LIN {X 0,Y 446.461,Z 349.006,A -85,B 0,C 180,E1 -8845.153,E2 -8845.153} C_VEL
LIN {X 0,Y 446.623,Z 343.213,A -85,B 0,C 180,E1 -8848.209,E2 -8848.209} C_VEL
LIN {X 0,Y 446.792,Z 337.441,A -85,B 0,C 180,E1 -8851.271,E2 -8851.271} C_VEL
LIN {X 0,Y 446.944,Z 331.506,A -85,B 0,C 180,E1 -8854.478,E2 -8854.478} C_VEL
LIN {X 0,Y 446.761,Z 327.48,A -85,B 0,C 180,E1 -8856.711,E2 -8856.711} C_VEL
LIN {X 0,Y 446.448,Z 325.193,A -85,B 0,C 180,E1 -8858.083,E2 -8858.083} C_VEL
LIN {X 0,Y 446.427,Z 325.192,A -85,B 0,C 180,E1 -8861.392,E2 -8861.392} C_VEL
LIN {X 0,Y 446.459,Z 325.185,A -85,B 0,C 180,E1 -8865.103,E2 -8865.103} C_VEL
LIN {X 0,Y 446.427,Z 325.19,A -85,B 0,C 180,E1 -8868.607,E2 -8868.607} C_VEL
LIN {X 0,Y 446.446,Z 325.238,A -85,B 0,C 180,E1 -8872.195,E2 -8872.195} C_VEL
LIN {X 0,Y 447.33,Z 330.595,A -85,B 0,C 180,E1 -8874.456,E2 -8874.456} C_VEL
LIN {X 0,Y 447.36,Z 335.572,A -85,B 0,C 180,E1 -8876.642,E2 -8876.642} C_VEL
LIN {X 0,Y 447.289,Z 341.416,A -85,B 0,C 180,E1 -8879.291,E2 -8879.291} C_VEL
LIN {X 0,Y 447.134,Z 348.904,A -85,B 0,C 180,E1 -8882.881,E2 -8882.881} C_VEL
LIN {X 0,Y 447.053,Z 356.132,A -85,B 0,C 180,E1 -8886.365,E2 -8886.365} C_VEL
LIN {X 0,Y 447.035,Z 362.429,A -85,B 0,C 180,E1 -8889.282,E2 -8889.282} C_VEL
LIN {X 0,Y 447.062,Z 369.132,A -85,B 0,C 180,E1 -8892.147,E2 -8892.147} C_VEL
LIN {X 0,Y 447.15,Z 373.659,A -85,B 0,C 180,E1 -8893.935,E2 -8893.935} C_VEL
LIN {X 0,Y 450.462,Z 384.816,A -85,B 0,C 180,E1 -8894.365,E2 -8894.365} C_VEL
LIN {X 0,Y 450.278,Z 397.037,A -85,B 0,C 180,E1 -8894.843,E2 -8894.843} C_VEL
LIN {X 0,Y 450.162,Z 402.389,A -85,B 0,C 180,E1 -8895.109,E2 -8895.109} C_VEL
LIN {X 0,Y 449.369,Z 407.874,A -85,B 0,C 180,E1 -8895.39,E2 -8895.39} C_VEL
LIN {X 0,Y 446.264,Z 416.577,A -85,B 0,C 180,E1 -8895.849,E2 -8895.849} C_VEL
LIN {X 0,Y 443.161,Z 424.955,A -85,B 0,C 180,E1 -8896.399,E2 -8896.399} C_VEL
LIN {X 0,Y 442.371,Z 429.793,A -85,B 0,C 180,E1 -8896.82,E2 -8896.82} C_VEL
LIN {X 0,Y 441.837,Z 439.223,A -85,B 0,C 180,E1 -8897.831,E2 -8897.831} C_VEL
LIN {X 0,Y 441.38,Z 447.936,A -85,B 0,C 180,E1 -8898.983,E2 -8898.983} C_VEL
LIN {X 0,Y 440.744,Z 456.447,A -85,B 0,C 180,E1 -8900.36,E2 -8900.36} C_VEL
LIN {X 0,Y 440.416,Z 463.236,A -85,B 0,C 180,E1 -8901.741,E2 -8901.741} C_VEL
LIN {X 0,Y 440.057,Z 468.639,A -85,B 0,C 180,E1 -8903.119,E2 -8903.119} C_VEL
LIN {X 0,Y 439.605,Z 472.902,A -85,B 0,C 180,E1 -8904.493,E2 -8904.493} C_VEL
LIN {X 0,Y 439.523,Z 475.12,A -85,B 0,C 180,E1 -8905.412,E2 -8905.412} C_VEL
LIN {X 0,Y 439.525,Z 476.919,A -85,B 0,C 180,E1 -8906.331,E2 -8906.331} C_VEL
LIN {X 0,Y 439.382,Z 478.317,A -85,B 0,C 180,E1 -8907.247,E2 -8907.247} C_VEL
LIN {X 0,Y 439.289,Z 479.89,A -85,B 0,C 180,E1 -8909.081,E2 -8909.081} C_VEL
LIN {X 0,Y 439.262,Z 480.124,A -85,B 0,C 180,E1 -8909.998,E2 -8909.998} C_VEL
LIN {X 0,Y 439.328,Z 479.368,A -85,B 0,C 180,E1 -8911.831,E2 -8911.831} C_VEL
LIN {X 0,Y 439.568,Z 477.087,A -85,B 0,C 180,E1 -8913.664,E2 -8913.664} C_VEL
LIN {X 0,Y 439.664,Z 474.304,A -85,B 0,C 180,E1 -8915.041,E2 -8915.041} C_VEL
LIN {X 0,Y 439.899,Z 470.504,A -85,B 0,C 180,E1 -8916.419,E2 -8916.419} C_VEL
LIN {X 0,Y 440.256,Z 465.229,A -85,B 0,C 180,E1 -8917.878,E2 -8917.878} C_VEL
LIN {X 0,Y 440.681,Z 458.173,A -85,B 0,C 180,E1 -8919.406,E2 -8919.406} C_VEL
LIN {X 0,Y 441.253,Z 450.147,A -85,B 0,C 180,E1 -8920.784,E2 -8920.784} C_VEL
LIN {X 0,Y 441.749,Z 441.869,A -85,B 0,C 180,E1 -8921.934,E2 -8921.934} C_VEL
LIN {X 0,Y 442.246,Z 431.688,A -85,B 0,C 180,E1 -8923.086,E2 -8923.086} C_VEL
LIN {X 0,Y 442.817,Z 421.179,A -85,B 0,C 180,E1 -8924.037,E2 -8924.037} C_VEL
LIN {X 0,Y 443.136,Z 410.38,A -85,B 0,C 180,E1 -8924.815,E2 -8924.815} C_VEL
LIN {X 0,Y 443.557,Z 397.678,A -85,B 0,C 180,E1 -8925.506,E2 -8925.506} C_VEL
LIN {X 0,Y 443.583,Z 385.861,A -85,B 0,C 180,E1 -8925.977,E2 -8925.977} C_VEL
LIN {X 0,Y 440.246,Z 374.666,A -85,B 0,C 180,E1 -8926.418,E2 -8926.418} C_VEL
LIN {X 0,Y 440.106,Z 366.794,A -85,B 0,C 180,E1 -8929.591,E2 -8929.591} C_VEL
LIN {X 0,Y 440.115,Z 359.098,A -85,B 0,C 180,E1 -8933.028,E2 -8933.028} C_VEL
LIN {X 0,Y 440.174,Z 351.628,A -85,B 0,C 180,E1 -8936.604,E2 -8936.604} C_VEL
LIN {X 0,Y 440.283,Z 345.234,A -85,B 0,C 180,E1 -8939.656,E2 -8939.656} C_VEL
LIN {X 0,Y 440.425,Z 338.39,A -85,B 0,C 180,E1 -8942.854,E2 -8942.854} C_VEL
LIN {X 0,Y 440.417,Z 332.314,A -85,B 0,C 180,E1 -8945.527,E2 -8945.527} C_VEL
LIN {X 0,Y 439.411,Z 326.272,A -85,B 0,C 180,E1 -8948.099,E2 -8948.099} C_VEL
LIN {X 0,Y 439.368,Z 326.07,A -85,B 0,C 180,E1 -8951.253,E2 -8951.253} C_VEL
LIN {X 0,Y 439.387,Z 326.066,A -85,B 0,C 180,E1 -8954.727,E2 -8954.727} C_VEL
LIN {X 0,Y 439.397,Z 326.062,A -85,B 0,C 180,E1 -8957.795,E2 -8957.795} C_VEL
LIN {X 0,Y 439.438,Z 326.06,A -85,B 0,C 180,E1 -8960.228,E2 -8960.228} C_VEL
LIN {X 0,Y 439.359,Z 326.071,A -85,B 0,C 180,E1 -8963.711,E2 -8963.711} C_VEL
LIN {X 0,Y 439.353,Z 326.069,A -85,B 0,C 180,E1 -8967.052,E2 -8967.052} C_VEL
LIN {X 0,Y 439.362,Z 326.064,A -85,B 0,C 180,E1 -8970.272,E2 -8970.272} C_VEL
LIN {X 0,Y 439.409,Z 326.056,A -85,B 0,C 180,E1 -8973.395,E2 -8973.395} C_VEL
LIN {X 0,Y 439.378,Z 326.063,A -85,B 0,C 180,E1 -8976.429,E2 -8976.429} C_VEL
LIN {X 0,Y 439.392,Z 326.067,A -85,B 0,C 180,E1 -8979.397,E2 -8979.397} C_VEL
LIN {X 0,Y 439.407,Z 326.059,A -85,B 0,C 180,E1 -8982.308,E2 -8982.308} C_VEL
LIN {X 0,Y 439.425,Z 326.054,A -85,B 0,C 180,E1 -8985.173,E2 -8985.173} C_VEL
LIN {X 0,Y 439.493,Z 326.052,A -85,B 0,C 180,E1 -8988.001,E2 -8988.001} C_VEL
LIN {X 0,Y 439.525,Z 326.045,A -85,B 0,C 180,E1 -8991.725,E2 -8991.725} C_VEL
LIN {X 0,Y 439.599,Z 326.034,A -85,B 0,C 180,E1 -8994.495,E2 -8994.495} C_VEL
LIN {X 0,Y 439.608,Z 326.037,A -85,B 0,C 180,E1 -8998.167,E2 -8998.167} C_VEL
LIN {X 0,Y 439.736,Z 326.017,A -85,B 0,C 180,E1 -9000,E2 -9000} C_VEL
LIN {X 0,Y 439.642,Z 326.034,A -85,B 0,C 180,E1 -9002.748,E2 -9002.748} C_VEL
LIN {X 0,Y 439.599,Z 326.037,A -85,B 0,C 180,E1 -9006.425,E2 -9006.425} C_VEL
LIN {X 0,Y 439.478,Z 326.056,A -85,B 0,C 180,E1 -9009.202,E2 -9009.202} C_VEL
LIN {X 0,Y 439.479,Z 326.057,A -85,B 0,C 180,E1 -9012.727,E2 -9012.727} C_VEL
LIN {X 0,Y 439.437,Z 326.062,A -85,B 0,C 180,E1 -9016.356,E2 -9016.356} C_VEL
LIN {X 0,Y 439.412,Z 326.065,A -85,B 0,C 180,E1 -9019.625,E2 -9019.625} C_VEL
LIN {X 0,Y 439.361,Z 326.068,A -85,B 0,C 180,E1 -9022.575,E2 -9022.575} C_VEL
LIN {X 0,Y 439.383,Z 326.065,A -85,B 0,C 180,E1 -9025.586,E2 -9025.586} C_VEL
LIN {X 0,Y 439.394,Z 326.066,A -85,B 0,C 180,E1 -9028.675,E2 -9028.675} C_VEL
LIN {X 0,Y 439.348,Z 326.072,A -85,B 0,C 180,E1 -9032.032,E2 -9032.032} C_VEL
LIN {X 0,Y 439.375,Z 326.069,A -85,B 0,C 180,E1 -9035.342,E2 -9035.342} C_VEL
LIN {X 0,Y 439.368,Z 326.069,A -85,B 0,C 180,E1 -9038.596,E2 -9038.596} C_VEL
LIN {X 0,Y 439.368,Z 326.062,A -85,B 0,C 180,E1 -9041.259,E2 -9041.259} C_VEL
LIN {X 0,Y 439.371,Z 326.248,A -85,B 0,C 180,E1 -9042.947,E2 -9042.947} C_VEL
LIN {X 0,Y 442.981,Z 337.856,A -85,B 0,C 180,E1 -9046.208,E2 -9046.208} C_VEL
LIN {X 0,Y 446.307,Z 349.009,A -85,B 0,C 180,E1 -9049.1,E2 -9049.1} C_VEL
LIN {X 0,Y 449.627,Z 361.072,A -85,B 0,C 180,E1 -9051.982,E2 -9051.982} C_VEL
LIN {X 0,Y 450.25,Z 364.591,A -85,B 0,C 180,E1 -9052.755,E2 -9052.755} C_VEL
LIN {X 0,Y 448.272,Z 381.256,A -85,B 0,C 180,E1 -9055.841,E2 -9055.841} C_VEL
LIN {X 0,Y 446.343,Z 400.241,A -85,B 0,C 180,E1 -9059.224,E2 -9059.224} C_VEL
LIN {X 0,Y 444.714,Z 418.995,A -85,B 0,C 180,E1 -9062.434,E2 -9062.434} C_VEL
LIN {X 0,Y 448.564,Z 438.005,A -85,B 0,C 180,E1 -9063.026,E2 -9063.026} C_VEL
LIN {X 0,Y 450.842,Z 449.868,A -85,B 0,C 180,E1 -9063.456,E2 -9063.456} C_VEL
LIN {X 0,Y 450.018,Z 466.755,A -85,B 0,C 180,E1 -9064.027,E2 -9064.027} C_VEL
LIN {X 0,Y 448.92,Z 482.813,A -85,B 0,C 180,E1 -9064.751,E2 -9064.751} C_VEL
LIN {X 0,Y 447.777,Z 498.534,A -85,B 0,C 180,E1 -9065.655,E2 -9065.655} C_VEL
LIN {X 0,Y 446.46,Z 513.475,A -85,B 0,C 180,E1 -9066.705,E2 -9066.705} C_VEL
LIN {X 0,Y 445.229,Z 527.23,A -85,B 0,C 180,E1 -9067.863,E2 -9067.863} C_VEL
LIN {X 0,Y 443.946,Z 540.246,A -85,B 0,C 180,E1 -9069.164,E2 -9069.164} C_VEL
LIN {X 0,Y 442.819,Z 551.987,A -85,B 0,C 180,E1 -9070.534,E2 -9070.534} C_VEL
LIN {X 0,Y 441.677,Z 563.981,A -85,B 0,C 180,E1 -9072.166,E2 -9072.166} C_VEL
LIN {X 0,Y 440.861,Z 574.252,A -85,B 0,C 180,E1 -9073.804,E2 -9073.804} C_VEL
LIN {X 0,Y 439.913,Z 584.129,A -85,B 0,C 180,E1 -9075.666,E2 -9075.666} C_VEL
LIN {X 0,Y 439.314,Z 592.39,A -85,B 0,C 180,E1 -9077.521,E2 -9077.521} C_VEL
LIN {X 0,Y 438.849,Z 599.352,A -85,B 0,C 180,E1 -9079.39,E2 -9079.39} C_VEL
LIN {X 0,Y 438.557,Z 604.908,A -85,B 0,C 180,E1 -9081.246,E2 -9081.246} C_VEL
LIN {X 0,Y 438.487,Z 608.25,A -85,B 0,C 180,E1 -9082.636,E2 -9082.636} C_VEL
LIN {X 0,Y 438.325,Z 611.637,A -85,B 0,C 180,E1 -9084.482,E2 -9084.482} C_VEL
LIN {X 0,Y 438.232,Z 614.093,A -85,B 0,C 180,E1 -9086.324,E2 -9086.324} C_VEL
LIN {X 0,Y 438.267,Z 615.479,A -85,B 0,C 180,E1 -9088.164,E2 -9088.164} C_VEL
LIN {X 0,Y 438.201,Z 616,A -85,B 0,C 180,E1 -9090.002,E2 -9090.002} C_VEL
LIN {X 0,Y 438.268,Z 615.475,A -85,B 0,C 180,E1 -9091.84,E2 -9091.84} C_VEL
LIN {X 0,Y 438.233,Z 614.087,A -85,B 0,C 180,E1 -9093.68,E2 -9093.68} C_VEL
LIN {X 0,Y 438.328,Z 611.629,A -85,B 0,C 180,E1 -9095.523,E2 -9095.523} C_VEL
LIN {X 0,Y 438.491,Z 608.248,A -85,B 0,C 180,E1 -9097.369,E2 -9097.369} C_VEL
LIN {X 0,Y 438.61,Z 603.623,A -85,B 0,C 180,E1 -9099.222,E2 -9099.222} C_VEL
LIN {X 0,Y 438.95,Z 597.704,A -85,B 0,C 180,E1 -9101.079,E2 -9101.079} C_VEL
LIN {X 0,Y 439.462,Z 590.425,A -85,B 0,C 180,E1 -9102.94,E2 -9102.94} C_VEL
LIN {X 0,Y 440.115,Z 581.588,A -85,B 0,C 180,E1 -9104.805,E2 -9104.805} C_VEL
LIN {X 0,Y 440.914,Z 572.495,A -85,B 0,C 180,E1 -9106.437,E2 -9106.437} C_VEL
LIN {X 0,Y 441.815,Z 561.902,A -85,B 0,C 180,E1 -9108.072,E2 -9108.072} C_VEL
LIN {X 0,Y 442.998,Z 549.4,A -85,B 0,C 180,E1 -9109.704,E2 -9109.704} C_VEL
LIN {X 0,Y 444.234,Z 536.263,A -85,B 0,C 180,E1 -9111.155,E2 -9111.155} C_VEL
LIN {X 0,Y 445.561,Z 521.959,A -85,B 0,C 180,E1 -9112.491,E2 -9112.491} C_VEL
LIN {X 0,Y 446.849,Z 507.165,A -85,B 0,C 180,E1 -9113.646,E2 -9113.646} C_VEL
LIN {X 0,Y 448.088,Z 491.339,A -85,B 0,C 180,E1 -9114.666,E2 -9114.666} C_VEL
LIN {X 0,Y 449.103,Z 476.791,A -85,B 0,C 180,E1 -9115.429,E2 -9115.429} C_VEL
LIN {X 0,Y 449.967,Z 461.122,A -85,B 0,C 180,E1 -9116.073,E2 -9116.073} C_VEL
LIN {X 0,Y 450.451,Z 448.549,A -85,B 0,C 180,E1 -9116.483,E2 -9116.483} C_VEL
LIN {X 0,Y 446.474,Z 429.842,A -85,B 0,C 180,E1 -9117.127,E2 -9117.127} C_VEL
LIN {X 0,Y 444.442,Z 417.956,A -85,B 0,C 180,E1 -9117.482,E2 -9117.482} C_VEL
LIN {X 0,Y 445.968,Z 398.339,A -85,B 0,C 180,E1 -9120.81,E2 -9120.81} C_VEL
LIN {X 0,Y 447.911,Z 381.252,A -85,B 0,C 180,E1 -9123.963,E2 -9123.963} C_VEL
LIN {X 0,Y 449.866,Z 369.238,A -85,B 0,C 180,E1 -9126.418,E2 -9126.418} C_VEL
LIN {X 0,Y 450.593,Z 364.614,A -85,B 0,C 180,E1 -9127.468,E2 -9127.468} C_VEL
LIN {X 0,Y 449.805,Z 360.335,A -85,B 0,C 180,E1 -9128.683,E2 -9128.683} C_VEL
LIN {X 0,Y 448.275,Z 354.936,A -85,B 0,C 180,E1 -9130.543,E2 -9130.543} C_VEL
LIN {X 0,Y 446.832,Z 350.314,A -85,B 0,C 180,E1 -9132.559,E2 -9132.559} C_VEL
LIN {X 0,Y 445.545,Z 346.703,A -85,B 0,C 180,E1 -9134.78,E2 -9134.78} C_VEL
LIN {X 0,Y 444.874,Z 344.812,A -85,B 0,C 180,E1 -9136.612,E2 -9136.612} C_VEL
LIN {X 0,Y 444.45,Z 343.921,A -85,B 0,C 180,E1 -9138.384,E2 -9138.384} C_VEL
LIN {X 0,Y 444.133,Z 344.024,A -85,B 0,C 180,E1 -9140.731,E2 -9140.731} C_VEL
LIN {X 0,Y 444.01,Z 345.321,A -85,B 0,C 180,E1 -9143.024,E2 -9143.024} C_VEL
LIN {X 0,Y 443.891,Z 346.316,A -85,B 0,C 180,E1 -9144.14,E2 -9144.14} C_VEL
LIN {X 0,Y 443.269,Z 348.846,A -85,B 0,C 180,E1 -9146.295,E2 -9146.295} C_VEL
LIN {X 0,Y 442.41,Z 353.265,A -85,B 0,C 180,E1 -9149.447,E2 -9149.447} C_VEL
LIN {X 0,Y 441.782,Z 358.656,A -85,B 0,C 180,E1 -9152.984,E2 -9152.984} C_VEL
LIN {X 0,Y 441.41,Z 362.771,A -85,B 0,C 180,E1 -9155.546,E2 -9155.546} C_VEL
LIN {X 0,Y 441.086,Z 367.633,A -85,B 0,C 180,E1 -9158.502,E2 -9158.502} C_VEL
LIN {X 0,Y 440.69,Z 373.409,A -85,B 0,C 180,E1 -9161.882,E2 -9161.882} C_VEL
LIN {X 0,Y 440.661,Z 374.052,A -85,B 0,C 180,E1 -9162.26,E2 -9162.26} C_VEL
LIN {X 0,Y 445.876,Z 388.81,A -85,B 0,C 180,E1 -9163.25,E2 -9163.25} C_VEL
LIN {X 0,Y 446.258,Z 389.984,A -85,B 0,C 180,E1 -9163.332,E2 -9163.332} C_VEL
LIN {X 0,Y 445.506,Z 404.424,A -85,B 0,C 180,E1 -9164.133,E2 -9164.133} C_VEL
LIN {X 0,Y 444.724,Z 416.942,A -85,B 0,C 180,E1 -9165.017,E2 -9165.017} C_VEL
LIN {X 0,Y 443.894,Z 428.51,A -85,B 0,C 180,E1 -9166.028,E2 -9166.028} C_VEL
LIN {X 0,Y 443.133,Z 439.164,A -85,B 0,C 180,E1 -9167.172,E2 -9167.172} C_VEL
LIN {X 0,Y 442.528,Z 447.959,A -85,B 0,C 180,E1 -9168.318,E2 -9168.318} C_VEL
LIN {X 0,Y 441.789,Z 456.684,A -85,B 0,C 180,E1 -9169.691,E2 -9169.691} C_VEL
LIN {X 0,Y 441.224,Z 464.001,A -85,B 0,C 180,E1 -9171.124,E2 -9171.124} C_VEL
LIN {X 0,Y 440.591,Z 470.283,A -85,B 0,C 180,E1 -9172.669,E2 -9172.669} C_VEL
LIN {X 0,Y 440.281,Z 474.558,A -85,B 0,C 180,E1 -9174.045,E2 -9174.045} C_VEL
LIN {X 0,Y 440.078,Z 477.764,A -85,B 0,C 180,E1 -9175.42,E2 -9175.42} C_VEL
LIN {X 0,Y 439.939,Z 479.386,A -85,B 0,C 180,E1 -9176.337,E2 -9176.337} C_VEL
LIN {X 0,Y 439.781,Z 480.56,A -85,B 0,C 180,E1 -9177.252,E2 -9177.252} C_VEL
LIN {X 0,Y 439.59,Z 481.33,A -85,B 0,C 180,E1 -9178.168,E2 -9178.168} C_VEL
LIN {X 0,Y 439.525,Z 481.683,A -85,B 0,C 180,E1 -9179.084,E2 -9179.084} C_VEL
LIN {X 0,Y 439.45,Z 481.649,A -85,B 0,C 180,E1 -9180,E2 -9180} C_VEL
LIN {X 0,Y 439.413,Z 481.201,A -85,B 0,C 180,E1 -9180.917,E2 -9180.917} C_VEL
LIN {X 0,Y 439.416,Z 480.322,A -85,B 0,C 180,E1 -9181.833,E2 -9181.833} C_VEL
LIN {X 0,Y 439.518,Z 479.036,A -85,B 0,C 180,E1 -9182.75,E2 -9182.75} C_VEL
LIN {X 0,Y 439.509,Z 476.345,A -85,B 0,C 180,E1 -9184.127,E2 -9184.127} C_VEL
LIN {X 0,Y 439.516,Z 472.663,A -85,B 0,C 180,E1 -9185.506,E2 -9185.506} C_VEL
LIN {X 0,Y 439.883,Z 467.862,A -85,B 0,C 180,E1 -9186.883,E2 -9186.883} C_VEL
LIN {X 0,Y 440.15,Z 460.779,A -85,B 0,C 180,E1 -9188.494,E2 -9188.494} C_VEL
LIN {X 0,Y 440.59,Z 453.141,A -85,B 0,C 180,E1 -9189.874,E2 -9189.874} C_VEL
LIN {X 0,Y 440.995,Z 443.74,A -85,B 0,C 180,E1 -9191.258,E2 -9191.258} C_VEL
LIN {X 0,Y 441.643,Z 433.185,A -85,B 0,C 180,E1 -9192.523,E2 -9192.523} C_VEL
LIN {X 0,Y 442.18,Z 421.281,A -85,B 0,C 180,E1 -9193.676,E2 -9193.676} C_VEL
LIN {X 0,Y 442.714,Z 409.036,A -85,B 0,C 180,E1 -9194.632,E2 -9194.632} C_VEL
LIN {X 0,Y 443.317,Z 396.509,A -85,B 0,C 180,E1 -9195.399,E2 -9195.399} C_VEL
LIN {X 0,Y 443.526,Z 384.753,A -85,B 0,C 180,E1 -9195.969,E2 -9195.969} C_VEL
LIN {X 0,Y 440.231,Z 370.942,A -85,B 0,C 180,E1 -9196.607,E2 -9196.607} C_VEL
LIN {X 0,Y 439.07,Z 366.227,A -85,B 0,C 180,E1 -9196.806,E2 -9196.806} C_VEL
LIN {X 0,Y 439.16,Z 360.671,A -85,B 0,C 180,E1 -9199.638,E2 -9199.638} C_VEL
LIN {X 0,Y 439.289,Z 354.989,A -85,B 0,C 180,E1 -9202.58,E2 -9202.58} C_VEL
LIN {X 0,Y 439.444,Z 349.231,A -85,B 0,C 180,E1 -9205.583,E2 -9205.583} C_VEL
LIN {X 0,Y 439.617,Z 343.434,A -85,B 0,C 180,E1 -9208.66,E2 -9208.66} C_VEL
LIN {X 0,Y 439.838,Z 336.984,A -85,B 0,C 180,E1 -9212.125,E2 -9212.125} C_VEL
LIN {X 0,Y 439.939,Z 331.552,A -85,B 0,C 180,E1 -9215.107,E2 -9215.107} C_VEL
LIN {X 0,Y 439.605,Z 327.454,A -85,B 0,C 180,E1 -9217.41,E2 -9217.41} C_VEL
LIN {X 0,Y 439.403,Z 326.069,A -85,B 0,C 180,E1 -9218.314,E2 -9218.314} C_VEL
LIN {X 0,Y 439.39,Z 326.069,A -85,B 0,C 180,E1 -9221.255,E2 -9221.255} C_VEL
LIN {X 0,Y 439.407,Z 326.062,A -85,B 0,C 180,E1 -9224.729,E2 -9224.729} C_VEL
LIN {X 0,Y 439.393,Z 326.067,A -85,B 0,C 180,E1 -9227.793,E2 -9227.793} C_VEL
LIN {X 0,Y 439.367,Z 326.071,A -85,B 0,C 180,E1 -9230.219,E2 -9230.219} C_VEL
LIN {X 0,Y 439.424,Z 326.156,A -85,B 0,C 180,E1 -9231.944,E2 -9231.944} C_VEL
LIN {X 0,Y 440.38,Z 332.057,A -85,B 0,C 180,E1 -9234.48,E2 -9234.48} C_VEL
LIN {X 0,Y 440.377,Z 338.112,A -85,B 0,C 180,E1 -9237.137,E2 -9237.137} C_VEL
LIN {X 0,Y 440.289,Z 343.279,A -85,B 0,C 180,E1 -9239.538,E2 -9239.538} C_VEL
LIN {X 0,Y 440.169,Z 350.428,A -85,B 0,C 180,E1 -9242.931,E2 -9242.931} C_VEL
LIN {X 0,Y 440.101,Z 357.804,A -85,B 0,C 180,E1 -9246.468,E2 -9246.468} C_VEL
LIN {X 0,Y 440.095,Z 364.282,A -85,B 0,C 180,E1 -9249.43,E2 -9249.43} C_VEL
LIN {X 0,Y 440.132,Z 371.194,A -85,B 0,C 180,E1 -9252.337,E2 -9252.337} C_VEL
LIN {X 0,Y 440.23,Z 374.625,A -85,B 0,C 180,E1 -9253.67,E2 -9253.67} C_VEL
LIN {X 0,Y 443.722,Z 386.858,A -85,B 0,C 180,E1 -9254.157,E2 -9254.157} C_VEL
LIN {X 0,Y 443.505,Z 399.298,A -85,B 0,C 180,E1 -9254.664,E2 -9254.664} C_VEL
LIN {X 0,Y 443.097,Z 411.668,A -85,B 0,C 180,E1 -9255.36,E2 -9255.36} C_VEL
LIN {X 0,Y 442.665,Z 423.158,A -85,B 0,C 180,E1 -9256.221,E2 -9256.221} C_VEL
LIN {X 0,Y 442.371,Z 429.793,A -85,B 0,C 180,E1 -9256.82,E2 -9256.82} C_VEL
LIN {X 0,Y 441.605,Z 434.491,A -85,B 0,C 180,E1 -9257.273,E2 -9257.273} C_VEL
LIN {X 0,Y 438.52,Z 441.99,A -85,B 0,C 180,E1 -9258.014,E2 -9258.014} C_VEL
LIN {X 0,Y 435.241,Z 448.977,A -85,B 0,C 180,E1 -9258.832,E2 -9258.832} C_VEL
LIN {X 0,Y 434.191,Z 452.875,A -85,B 0,C 180,E1 -9259.403,E2 -9259.403} C_VEL
LIN {X 0,Y 433.717,Z 459.935,A -85,B 0,C 180,E1 -9260.673,E2 -9260.673} C_VEL
LIN {X 0,Y 433.282,Z 466.931,A -85,B 0,C 180,E1 -9262.244,E2 -9262.244} C_VEL
LIN {X 0,Y 432.947,Z 471.261,A -85,B 0,C 180,E1 -9263.473,E2 -9263.473} C_VEL
LIN {X 0,Y 432.663,Z 475.144,A -85,B 0,C 180,E1 -9264.872,E2 -9264.872} C_VEL
LIN {X 0,Y 432.529,Z 477.995,A -85,B 0,C 180,E1 -9266.271,E2 -9266.271} C_VEL
LIN {X 0,Y 432.401,Z 479.39,A -85,B 0,C 180,E1 -9267.203,E2 -9267.203} C_VEL
LIN {X 0,Y 432.275,Z 480.967,A -85,B 0,C 180,E1 -9269.066,E2 -9269.066} C_VEL
LIN {X 0,Y 432.245,Z 481.201,A -85,B 0,C 180,E1 -9269.998,E2 -9269.998} C_VEL
LIN {X 0,Y 432.325,Z 480.443,A -85,B 0,C 180,E1 -9271.861,E2 -9271.861} C_VEL
LIN {X 0,Y 432.566,Z 478.162,A -85,B 0,C 180,E1 -9273.724,E2 -9273.724} C_VEL
LIN {X 0,Y 432.671,Z 475.379,A -85,B 0,C 180,E1 -9275.123,E2 -9275.123} C_VEL
LIN {X 0,Y 432.929,Z 471.577,A -85,B 0,C 180,E1 -9276.522,E2 -9276.522} C_VEL
LIN {X 0,Y 433.322,Z 466.192,A -85,B 0,C 180,E1 -9278.031,E2 -9278.031} C_VEL
LIN {X 0,Y 433.755,Z 459.245,A -85,B 0,C 180,E1 -9279.557,E2 -9279.557} C_VEL
LIN {X 0,Y 434.369,Z 451.214,A -85,B 0,C 180,E1 -9280.957,E2 -9280.957} C_VEL
LIN {X 0,Y 434.889,Z 442.933,A -85,B 0,C 180,E1 -9282.125,E2 -9282.125} C_VEL
LIN {X 0,Y 435.427,Z 432.747,A -85,B 0,C 180,E1 -9283.295,E2 -9283.295} C_VEL
LIN {X 0,Y 436.018,Z 422.191,A -85,B 0,C 180,E1 -9284.264,E2 -9284.264} C_VEL
LIN {X 0,Y 436.347,Z 411.426,A -85,B 0,C 180,E1 -9285.051,E2 -9285.051} C_VEL
LIN {X 0,Y 436.782,Z 398.712,A -85,B 0,C 180,E1 -9285.752,E2 -9285.752} C_VEL
LIN {X 0,Y 436.914,Z 387.614,A -85,B 0,C 180,E1 -9286.201,E2 -9286.201} C_VEL
LIN {X 0,Y 433.337,Z 375.627,A -85,B 0,C 180,E1 -9286.696,E2 -9286.696} C_VEL
LIN {X 0,Y 433.186,Z 367.618,A -85,B 0,C 180,E1 -9289.917,E2 -9289.917} C_VEL
LIN {X 0,Y 433.167,Z 359.766,A -85,B 0,C 180,E1 -9293.419,E2 -9293.419} C_VEL
LIN {X 0,Y 433.21,Z 352.242,A -85,B 0,C 180,E1 -9297.013,E2 -9297.013} C_VEL
LIN {X 0,Y 433.346,Z 345.558,A -85,B 0,C 180,E1 -9300.179,E2 -9300.179} C_VEL
LIN {X 0,Y 433.488,Z 338.514,A -85,B 0,C 180,E1 -9303.448,E2 -9303.448} C_VEL
LIN {X 0,Y 433.386,Z 333.134,A -85,B 0,C 180,E1 -9305.823,E2 -9305.823} C_VEL
LIN {X 0,Y 432.456,Z 327.729,A -85,B 0,C 180,E1 -9308.134,E2 -9308.134} C_VEL
LIN {X 0,Y 432.321,Z 326.949,A -85,B 0,C 180,E1 -9308.514,E2 -9308.514} C_VEL
LIN {X 0,Y 432.31,Z 326.949,A -85,B 0,C 180,E1 -9311.796,E2 -9311.796} C_VEL
LIN {X 0,Y 432.364,Z 326.94,A -85,B 0,C 180,E1 -9315.656,E2 -9315.656} C_VEL
LIN {X 0,Y 432.358,Z 326.942,A -85,B 0,C 180,E1 -9318.389,E2 -9318.389} C_VEL
LIN {X 0,Y 432.338,Z 326.943,A -85,B 0,C 180,E1 -9321.85,E2 -9321.85} C_VEL
LIN {X 0,Y 432.322,Z 326.946,A -85,B 0,C 180,E1 -9325.321,E2 -9325.321} C_VEL
LIN {X 0,Y 432.301,Z 326.949,A -85,B 0,C 180,E1 -9328.652,E2 -9328.652} C_VEL
LIN {X 0,Y 432.362,Z 326.94,A -85,B 0,C 180,E1 -9331.875,E2 -9331.875} C_VEL
LIN {X 0,Y 432.338,Z 326.943,A -85,B 0,C 180,E1 -9334.998,E2 -9334.998} C_VEL
LIN {X 0,Y 432.389,Z 326.937,A -85,B 0,C 180,E1 -9338.047,E2 -9338.047} C_VEL
LIN {X 0,Y 432.363,Z 326.937,A -85,B 0,C 180,E1 -9341.028,E2 -9341.028} C_VEL
LIN {X 0,Y 432.407,Z 326.933,A -85,B 0,C 180,E1 -9343.96,E2 -9343.96} C_VEL
LIN {X 0,Y 432.464,Z 326.927,A -85,B 0,C 180,E1 -9347.803,E2 -9347.803} C_VEL
LIN {X 0,Y 432.469,Z 326.922,A -85,B 0,C 180,E1 -9351.59,E2 -9351.59} C_VEL
LIN {X 0,Y 432.575,Z 326.909,A -85,B 0,C 180,E1 -9354.405,E2 -9354.405} C_VEL
LIN {X 0,Y 432.577,Z 326.912,A -85,B 0,C 180,E1 -9358.138,E2 -9358.138} C_VEL
LIN {X 0,Y 432.706,Z 326.893,A -85,B 0,C 180,E1 -9360,E2 -9360} C_VEL
LIN {X 0,Y 432.592,Z 326.912,A -85,B 0,C 180,E1 -9362.793,E2 -9362.793} C_VEL
LIN {X 0,Y 432.552,Z 326.914,A -85,B 0,C 180,E1 -9366.53,E2 -9366.53} C_VEL
LIN {X 0,Y 432.422,Z 326.936,A -85,B 0,C 180,E1 -9369.353,E2 -9369.353} C_VEL
LIN {X 0,Y 432.419,Z 326.936,A -85,B 0,C 180,E1 -9372.812,E2 -9372.812} C_VEL
LIN {X 0,Y 432.399,Z 326.937,A -85,B 0,C 180,E1 -9376.485,E2 -9376.485} C_VEL
LIN {X 0,Y 432.359,Z 326.942,A -85,B 0,C 180,E1 -9379.959,E2 -9379.959} C_VEL
LIN {X 0,Y 432.31,Z 326.948,A -85,B 0,C 180,E1 -9382.964,E2 -9382.964} C_VEL
LIN {X 0,Y 432.341,Z 326.942,A -85,B 0,C 180,E1 -9386.034,E2 -9386.034} C_VEL
LIN {X 0,Y 432.319,Z 326.945,A -85,B 0,C 180,E1 -9389.189,E2 -9389.189} C_VEL
LIN {X 0,Y 432.301,Z 326.95,A -85,B 0,C 180,E1 -9392.444,E2 -9392.444} C_VEL
LIN {X 0,Y 432.325,Z 326.947,A -85,B 0,C 180,E1 -9395.634,E2 -9395.634} C_VEL
LIN {X 0,Y 432.331,Z 326.945,A -85,B 0,C 180,E1 -9398.718,E2 -9398.718} C_VEL
LIN {X 0,Y 432.356,Z 326.989,A -85,B 0,C 180,E1 -9402.186,E2 -9402.186} C_VEL
LIN {X 0,Y 436.303,Z 340.009,A -85,B 0,C 180,E1 -9405.924,E2 -9405.924} C_VEL
LIN {X 0,Y 439.476,Z 350.623,A -85,B 0,C 180,E1 -9408.73,E2 -9408.73} C_VEL
LIN {X 0,Y 442.95,Z 363.118,A -85,B 0,C 180,E1 -9411.776,E2 -9411.776} C_VEL
LIN {X 0,Y 443.582,Z 366.816,A -85,B 0,C 180,E1 -9412.606,E2 -9412.606} C_VEL
LIN {X 0,Y 441.61,Z 382.484,A -85,B 0,C 180,E1 -9415.565,E2 -9415.565} C_VEL
LIN {X 0,Y 439.679,Z 399.756,A -85,B 0,C 180,E1 -9418.705,E2 -9418.705} C_VEL
LIN {X 0,Y 437.968,Z 418.244,A -85,B 0,C 180,E1 -9421.954,E2 -9421.954} C_VEL
LIN {X 0,Y 437.938,Z 418.769,A -85,B 0,C 180,E1 -9422.039,E2 -9422.039} C_VEL
LIN {X 0,Y 442.163,Z 439.816,A -85,B 0,C 180,E1 -9422.713,E2 -9422.713} C_VEL
LIN {X 0,Y 444.247,Z 450.914,A -85,B 0,C 180,E1 -9423.142,E2 -9423.142} C_VEL
LIN {X 0,Y 443.356,Z 467.342,A -85,B 0,C 180,E1 -9423.717,E2 -9423.717} C_VEL
LIN {X 0,Y 442.213,Z 483.385,A -85,B 0,C 180,E1 -9424.466,E2 -9424.466} C_VEL
LIN {X 0,Y 441.037,Z 498.747,A -85,B 0,C 180,E1 -9425.377,E2 -9425.377} C_VEL
LIN {X 0,Y 439.66,Z 513.596,A -85,B 0,C 180,E1 -9426.448,E2 -9426.448} C_VEL
LIN {X 0,Y 438.249,Z 528.407,A -85,B 0,C 180,E1 -9427.74,E2 -9427.74} C_VEL
LIN {X 0,Y 436.881,Z 541.658,A -85,B 0,C 180,E1 -9429.11,E2 -9429.11} C_VEL
LIN {X 0,Y 435.605,Z 554.514,A -85,B 0,C 180,E1 -9430.689,E2 -9430.689} C_VEL
LIN {X 0,Y 434.504,Z 565.789,A -85,B 0,C 180,E1 -9432.319,E2 -9432.319} C_VEL
LIN {X 0,Y 433.649,Z 575.801,A -85,B 0,C 180,E1 -9434.01,E2 -9434.01} C_VEL
LIN {X 0,Y 432.73,Z 585.335,A -85,B 0,C 180,E1 -9435.903,E2 -9435.903} C_VEL
LIN {X 0,Y 432.151,Z 593.307,A -85,B 0,C 180,E1 -9437.797,E2 -9437.797} C_VEL
LIN {X 0,Y 431.672,Z 599.854,A -85,B 0,C 180,E1 -9439.686,E2 -9439.686} C_VEL
LIN {X 0,Y 431.478,Z 605.236,A -85,B 0,C 180,E1 -9441.573,E2 -9441.573} C_VEL
LIN {X 0,Y 431.321,Z 609.872,A -85,B 0,C 180,E1 -9443.687,E2 -9443.687} C_VEL
LIN {X 0,Y 431.211,Z 612.499,A -85,B 0,C 180,E1 -9445.328,E2 -9445.328} C_VEL
LIN {X 0,Y 431.196,Z 614.537,A -85,B 0,C 180,E1 -9447.2,E2 -9447.2} C_VEL
LIN {X 0,Y 431.144,Z 615.545,A -85,B 0,C 180,E1 -9449.068,E2 -9449.068} C_VEL
LIN {X 0,Y 431.144,Z 615.543,A -85,B 0,C 180,E1 -9450.936,E2 -9450.936} C_VEL
LIN {X 0,Y 431.197,Z 614.528,A -85,B 0,C 180,E1 -9452.805,E2 -9452.805} C_VEL
LIN {X 0,Y 431.213,Z 612.475,A -85,B 0,C 180,E1 -9454.676,E2 -9454.676} C_VEL
LIN {X 0,Y 431.362,Z 609.364,A -85,B 0,C 180,E1 -9456.551,E2 -9456.551} C_VEL
LIN {X 0,Y 431.48,Z 605.152,A -85,B 0,C 180,E1 -9458.432,E2 -9458.432} C_VEL
LIN {X 0,Y 431.681,Z 599.705,A -85,B 0,C 180,E1 -9460.319,E2 -9460.319} C_VEL
LIN {X 0,Y 432.186,Z 593.071,A -85,B 0,C 180,E1 -9462.206,E2 -9462.206} C_VEL
LIN {X 0,Y 432.755,Z 584.97,A -85,B 0,C 180,E1 -9464.101,E2 -9464.101} C_VEL
LIN {X 0,Y 433.645,Z 575.275,A -85,B 0,C 180,E1 -9465.995,E2 -9465.995} C_VEL
LIN {X 0,Y 434.466,Z 565.057,A -85,B 0,C 180,E1 -9467.686,E2 -9467.686} C_VEL
LIN {X 0,Y 435.58,Z 553.533,A -85,B 0,C 180,E1 -9469.317,E2 -9469.317} C_VEL
LIN {X 0,Y 436.873,Z 540.446,A -85,B 0,C 180,E1 -9470.889,E2 -9470.889} C_VEL
LIN {X 0,Y 438.186,Z 526.797,A -85,B 0,C 180,E1 -9472.269,E2 -9472.269} C_VEL
LIN {X 0,Y 439.407,Z 513.028,A -85,B 0,C 180,E1 -9473.446,E2 -9473.446} C_VEL
LIN {X 0,Y 440.797,Z 497.2,A -85,B 0,C 180,E1 -9474.572,E2 -9474.572} C_VEL
LIN {X 0,Y 442.003,Z 481.35,A -85,B 0,C 180,E1 -9475.489,E2 -9475.489} C_VEL
LIN {X 0,Y 443.027,Z 465.567,A -85,B 0,C 180,E1 -9476.214,E2 -9476.214} C_VEL
LIN {X 0,Y 443.827,Z 450.008,A -85,B 0,C 180,E1 -9476.755,E2 -9476.755} C_VEL
LIN {X 0,Y 440.208,Z 432.566,A -85,B 0,C 180,E1 -9477.401,E2 -9477.401} C_VEL
LIN {X 0,Y 437.6,Z 417.592,A -85,B 0,C 180,E1 -9477.858,E2 -9477.858} C_VEL
LIN {X 0,Y 439.182,Z 399.211,A -85,B 0,C 180,E1 -9481.071,E2 -9481.071} C_VEL
LIN {X 0,Y 441.14,Z 383.445,A -85,B 0,C 180,E1 -9484.062,E2 -9484.062} C_VEL
LIN {X 0,Y 443.635,Z 369.506,A -85,B 0,C 180,E1 -9487.014,E2 -9487.014} C_VEL
LIN {X 0,Y 443.966,Z 366.752,A -85,B 0,C 180,E1 -9487.674,E2 -9487.674} C_VEL
LIN {X 0,Y 443.088,Z 362.344,A -85,B 0,C 180,E1 -9488.995,E2 -9488.995} C_VEL
LIN {X 0,Y 441.74,Z 357.562,A -85,B 0,C 180,E1 -9490.717,E2 -9490.717} C_VEL
LIN {X 0,Y 440.327,Z 353.07,A -85,B 0,C 180,E1 -9492.761,E2 -9492.761} C_VEL
LIN {X 0,Y 439.195,Z 349.885,A -85,B 0,C 180,E1 -9494.758,E2 -9494.758} C_VEL
LIN {X 0,Y 438.542,Z 348.055,A -85,B 0,C 180,E1 -9496.441,E2 -9496.441} C_VEL
LIN {X 0,Y 438.2,Z 347.243,A -85,B 0,C 180,E1 -9497.654,E2 -9497.654} C_VEL
LIN {X 0,Y 437.717,Z 346.791,A -85,B 0,C 180,E1 -9500.041,E2 -9500.041} C_VEL
LIN {X 0,Y 437.507,Z 347.599,A -85,B 0,C 180,E1 -9502.38,E2 -9502.38} C_VEL
LIN {X 0,Y 437.106,Z 349.437,A -85,B 0,C 180,E1 -9504.632,E2 -9504.632} C_VEL
LIN {X 0,Y 436.382,Z 352.037,A -85,B 0,C 180,E1 -9506.876,E2 -9506.876} C_VEL
LIN {X 0,Y 435.378,Z 357.244,A -85,B 0,C 180,E1 -9510.657,E2 -9510.657} C_VEL
LIN {X 0,Y 434.941,Z 360.882,A -85,B 0,C 180,E1 -9513.1,E2 -9513.1} C_VEL
LIN {X 0,Y 434.458,Z 365.669,A -85,B 0,C 180,E1 -9516.146,E2 -9516.146} C_VEL
LIN {X 0,Y 434.143,Z 370.539,A -85,B 0,C 180,E1 -9519.137,E2 -9519.137} C_VEL
LIN {X 0,Y 433.83,Z 375.1,A -85,B 0,C 180,E1 -9521.813,E2 -9521.813} C_VEL
LIN {X 0,Y 438.73,Z 388.37,A -85,B 0,C 180,E1 -9522.751,E2 -9522.751} C_VEL
LIN {X 0,Y 439.801,Z 392.243,A -85,B 0,C 180,E1 -9523.027,E2 -9523.027} C_VEL
LIN {X 0,Y 438.926,Z 407.104,A -85,B 0,C 180,E1 -9523.889,E2 -9523.889} C_VEL
LIN {X 0,Y 438.183,Z 418.024,A -85,B 0,C 180,E1 -9524.687,E2 -9524.687} C_VEL
LIN {X 0,Y 437.241,Z 430.479,A -85,B 0,C 180,E1 -9525.811,E2 -9525.811} C_VEL
LIN {X 0,Y 436.434,Z 440.956,A -85,B 0,C 180,E1 -9526.971,E2 -9526.971} C_VEL
LIN {X 0,Y 435.789,Z 449.66,A -85,B 0,C 180,E1 -9528.135,E2 -9528.135} C_VEL
LIN {X 0,Y 434.993,Z 458.259,A -85,B 0,C 180,E1 -9529.528,E2 -9529.528} C_VEL
LIN {X 0,Y 434.315,Z 466.258,A -85,B 0,C 180,E1 -9531.157,E2 -9531.157} C_VEL
LIN {X 0,Y 433.697,Z 471.72,A -85,B 0,C 180,E1 -9532.552,E2 -9532.552} C_VEL
LIN {X 0,Y 433.383,Z 475.951,A -85,B 0,C 180,E1 -9533.95,E2 -9533.95} C_VEL
LIN {X 0,Y 433.156,Z 479.115,A -85,B 0,C 180,E1 -9535.347,E2 -9535.347} C_VEL
LIN {X 0,Y 432.983,Z 480.705,A -85,B 0,C 180,E1 -9536.278,E2 -9536.278} C_VEL
LIN {X 0,Y 432.827,Z 481.84,A -85,B 0,C 180,E1 -9537.208,E2 -9537.208} C_VEL
LIN {X 0,Y 432.626,Z 482.578,A -85,B 0,C 180,E1 -9538.138,E2 -9538.138} C_VEL
LIN {X 0,Y 432.548,Z 482.908,A -85,B 0,C 180,E1 -9539.069,E2 -9539.069} C_VEL
LIN {X 0,Y 432.474,Z 482.85,A -85,B 0,C 180,E1 -9540,E2 -9540} C_VEL
LIN {X 0,Y 432.421,Z 482.371,A -85,B 0,C 180,E1 -9540.932,E2 -9540.932} C_VEL
LIN {X 0,Y 432.413,Z 481.468,A -85,B 0,C 180,E1 -9541.863,E2 -9541.863} C_VEL
LIN {X 0,Y 432.522,Z 480.143,A -85,B 0,C 180,E1 -9542.794,E2 -9542.794} C_VEL
LIN {X 0,Y 432.505,Z 477.407,A -85,B 0,C 180,E1 -9544.194,E2 -9544.194} C_VEL
LIN {X 0,Y 432.522,Z 473.666,A -85,B 0,C 180,E1 -9545.595,E2 -9545.595} C_VEL
LIN {X 0,Y 432.909,Z 468.8,A -85,B 0,C 180,E1 -9546.994,E2 -9546.994} C_VEL
LIN {X 0,Y 433.2,Z 461.633,A -85,B 0,C 180,E1 -9548.631,E2 -9548.631} C_VEL
LIN {X 0,Y 433.664,Z 453.919,A -85,B 0,C 180,E1 -9550.033,E2 -9550.033} C_VEL
LIN {X 0,Y 434.08,Z 444.457,A -85,B 0,C 180,E1 -9551.44,E2 -9551.44} C_VEL
LIN {X 0,Y 434.753,Z 433.834,A -85,B 0,C 180,E1 -9552.724,E2 -9552.724} C_VEL
LIN {X 0,Y 435.321,Z 421.868,A -85,B 0,C 180,E1 -9553.896,E2 -9553.896} C_VEL
LIN {X 0,Y 435.87,Z 409.643,A -85,B 0,C 180,E1 -9554.863,E2 -9554.863} C_VEL
LIN {X 0,Y 436.517,Z 397.04,A -85,B 0,C 180,E1 -9555.645,E2 -9555.645} C_VEL
LIN {X 0,Y 436.699,Z 386.028,A -85,B 0,C 180,E1 -9556.195,E2 -9556.195} C_VEL
LIN {X 0,Y 433.44,Z 372.182,A -85,B 0,C 180,E1 -9556.85,E2 -9556.85} C_VEL
LIN {X 0,Y 432.041,Z 366.611,A -85,B 0,C 180,E1 -9557.087,E2 -9557.087} C_VEL
LIN {X 0,Y 432.137,Z 361.016,A -85,B 0,C 180,E1 -9559.971,E2 -9559.971} C_VEL
LIN {X 0,Y 432.26,Z 355.25,A -85,B 0,C 180,E1 -9562.968,E2 -9562.968} C_VEL
LIN {X 0,Y 432.427,Z 349.449,A -85,B 0,C 180,E1 -9566.029,E2 -9566.029} C_VEL
LIN {X 0,Y 432.618,Z 343.596,A -85,B 0,C 180,E1 -9569.168,E2 -9569.168} C_VEL
LIN {X 0,Y 432.845,Z 337.633,A -85,B 0,C 180,E1 -9572.4,E2 -9572.4} C_VEL
LIN {X 0,Y 432.931,Z 333.601,A -85,B 0,C 180,E1 -9574.623,E2 -9574.623} C_VEL
LIN {X 0,Y 432.73,Z 329.508,A -85,B 0,C 180,E1 -9576.936,E2 -9576.936} C_VEL
LIN {X 0,Y 432.356,Z 326.947,A -85,B 0,C 180,E1 -9578.429,E2 -9578.429} C_VEL
LIN {X 0,Y 432.333,Z 326.947,A -85,B 0,C 180,E1 -9581.798,E2 -9581.798} C_VEL
LIN {X 0,Y 432.343,Z 326.943,A -85,B 0,C 180,E1 -9584.347,E2 -9584.347} C_VEL
LIN {X 0,Y 432.325,Z 326.948,A -85,B 0,C 180,E1 -9587.016,E2 -9587.016} C_VEL
LIN {X 0,Y 432.322,Z 326.947,A -85,B 0,C 180,E1 -9589.823,E2 -9589.823} C_VEL
LIN {X 0,Y 432.38,Z 327.105,A -85,B 0,C 180,E1 -9591.713,E2 -9591.713} C_VEL
LIN {X 0,Y 433.369,Z 333.038,A -85,B 0,C 180,E1 -9594.279,E2 -9594.279} C_VEL
LIN {X 0,Y 433.502,Z 336.485,A -85,B 0,C 180,E1 -9595.774,E2 -9595.774} C_VEL
LIN {X 0,Y 433.412,Z 342.996,A -85,B 0,C 180,E1 -9598.74,E2 -9598.74} C_VEL
LIN {X 0,Y 433.238,Z 350.891,A -85,B 0,C 180,E1 -9602.461,E2 -9602.461} C_VEL
LIN {X 0,Y 433.131,Z 358.441,A -85,B 0,C 180,E1 -9606.066,E2 -9606.066} C_VEL
LIN {X 0,Y 433.151,Z 365.059,A -85,B 0,C 180,E1 -9609.085,E2 -9609.085} C_VEL
LIN {X 0,Y 433.202,Z 372.111,A -85,B 0,C 180,E1 -9612.045,E2 -9612.045} C_VEL
LIN {X 0,Y 433.308,Z 375.623,A -85,B 0,C 180,E1 -9613.405,E2 -9613.405} C_VEL
LIN {X 0,Y 436.968,Z 388.306,A -85,B 0,C 180,E1 -9613.92,E2 -9613.92} C_VEL
LIN {X 0,Y 436.676,Z 401.571,A -85,B 0,C 180,E1 -9614.478,E2 -9614.478} C_VEL
LIN {X 0,Y 436.33,Z 412.501,A -85,B 0,C 180,E1 -9615.112,E2 -9615.112} C_VEL
LIN {X 0,Y 435.85,Z 424.225,A -85,B 0,C 180,E1 -9616.001,E2 -9616.001} C_VEL
LIN {X 0,Y 435.339,Z 435.163,A -85,B 0,C 180,E1 -9617.054,E2 -9617.054} C_VEL
LIN {X 0,Y 434.848,Z 443.998,A -85,B 0,C 180,E1 -9618.106,E2 -9618.106} C_VEL
LIN {X 0,Y 434.191,Z 452.875,A -85,B 0,C 180,E1 -9619.403,E2 -9619.403} C_VEL
LIN {X 0,Y 433.188,Z 456.61,A -85,B 0,C 180,E1 -9620,E2 -9620} C_VEL
LIN {X 0,Y 430.058,Z 462.392,A -85,B 0,C 180,E1 -9620.988,E2 -9620.988} C_VEL
LIN {X 0,Y 427.027,Z 467.558,A -85,B 0,C 180,E1 -9622.041,E2 -9622.041} C_VEL
LIN {X 0,Y 426.186,Z 470.229,A -85,B 0,C 180,E1 -9622.735,E2 -9622.735} C_VEL
LIN {X 0,Y 425.635,Z 475.057,A -85,B 0,C 180,E1 -9624.312,E2 -9624.312} C_VEL
LIN {X 0,Y 425.536,Z 477.275,A -85,B 0,C 180,E1 -9625.261,E2 -9625.261} C_VEL
LIN {X 0,Y 425.532,Z 479.072,A -85,B 0,C 180,E1 -9626.21,E2 -9626.21} C_VEL
LIN {X 0,Y 425.416,Z 480.463,A -85,B 0,C 180,E1 -9627.157,E2 -9627.157} C_VEL
LIN {X 0,Y 425.26,Z 482.044,A -85,B 0,C 180,E1 -9629.051,E2 -9629.051} C_VEL
LIN {X 0,Y 425.228,Z 482.278,A -85,B 0,C 180,E1 -9629.998,E2 -9629.998} C_VEL
LIN {X 0,Y 425.321,Z 481.518,A -85,B 0,C 180,E1 -9631.892,E2 -9631.892} C_VEL
LIN {X 0,Y 425.563,Z 479.238,A -85,B 0,C 180,E1 -9633.785,E2 -9633.785} C_VEL
LIN {X 0,Y 425.68,Z 476.454,A -85,B 0,C 180,E1 -9635.208,E2 -9635.208} C_VEL
LIN {X 0,Y 425.96,Z 472.651,A -85,B 0,C 180,E1 -9636.63,E2 -9636.63} C_VEL
LIN {X 0,Y 426.392,Z 467.157,A -85,B 0,C 180,E1 -9638.189,E2 -9638.189} C_VEL
LIN {X 0,Y 426.834,Z 460.316,A -85,B 0,C 180,E1 -9639.714,E2 -9639.714} C_VEL
LIN {X 0,Y 427.505,Z 452.278,A -85,B 0,C 180,E1 -9641.135,E2 -9641.135} C_VEL
LIN {X 0,Y 428.03,Z 443.998,A -85,B 0,C 180,E1 -9642.322,E2 -9642.322} C_VEL
LIN {X 0,Y 428.614,Z 433.806,A -85,B 0,C 180,E1 -9643.51,E2 -9643.51} C_VEL
LIN {X 0,Y 429.224,Z 423.152,A -85,B 0,C 180,E1 -9644.502,E2 -9644.502} C_VEL
LIN {X 0,Y 429.583,Z 412.47,A -85,B 0,C 180,E1 -9645.293,E2 -9645.293} C_VEL
LIN {X 0,Y 430.024,Z 399.745,A -85,B 0,C 180,E1 -9646.007,E2 -9646.007} C_VEL
LIN {X 0,Y 430.049,Z 388.739,A -85,B 0,C 180,E1 -9646.463,E2 -9646.463} C_VEL
LIN {X 0,Y 426.415,Z 376.604,A -85,B 0,C 180,E1 -9646.979,E2 -9646.979} C_VEL
LIN {X 0,Y 426.239,Z 368.446,A -85,B 0,C 180,E1 -9650.256,E2 -9650.256} C_VEL
LIN {X 0,Y 426.228,Z 361.535,A -85,B 0,C 180,E1 -9653.309,E2 -9653.309} C_VEL
LIN {X 0,Y 426.254,Z 354.915,A -85,B 0,C 180,E1 -9656.431,E2 -9656.431} C_VEL
LIN {X 0,Y 426.36,Z 348.195,A -85,B 0,C 180,E1 -9659.634,E2 -9659.634} C_VEL
LIN {X 0,Y 426.528,Z 341.094,A -85,B 0,C 180,E1 -9662.936,E2 -9662.936} C_VEL
LIN {X 0,Y 426.5,Z 334.967,A -85,B 0,C 180,E1 -9665.666,E2 -9665.666} C_VEL
LIN {X 0,Y 425.773,Z 330.462,A -85,B 0,C 180,E1 -9667.639,E2 -9667.639} C_VEL
LIN {X 0,Y 425.274,Z 327.826,A -85,B 0,C 180,E1 -9668.821,E2 -9668.821} C_VEL
LIN {X 0,Y 425.269,Z 327.826,A -85,B 0,C 180,E1 -9671.954,E2 -9671.954} C_VEL
LIN {X 0,Y 425.299,Z 327.824,A -85,B 0,C 180,E1 -9675.277,E2 -9675.277} C_VEL
LIN {X 0,Y 425.295,Z 327.824,A -85,B 0,C 180,E1 -9678.623,E2 -9678.623} C_VEL
LIN {X 0,Y 425.31,Z 327.818,A -85,B 0,C 180,E1 -9681.102,E2 -9681.102} C_VEL
LIN {X 0,Y 425.282,Z 327.821,A -85,B 0,C 180,E1 -9684.662,E2 -9684.662} C_VEL
LIN {X 0,Y 425.245,Z 327.827,A -85,B 0,C 180,E1 -9688.071,E2 -9688.071} C_VEL
LIN {X 0,Y 425.311,Z 327.82,A -85,B 0,C 180,E1 -9691.366,E2 -9691.366} C_VEL
LIN {X 0,Y 425.281,Z 327.824,A -85,B 0,C 180,E1 -9694.553,E2 -9694.553} C_VEL
LIN {X 0,Y 425.307,Z 327.815,A -85,B 0,C 180,E1 -9697.715,E2 -9697.715} C_VEL
LIN {X 0,Y 425.342,Z 327.811,A -85,B 0,C 180,E1 -9700.703,E2 -9700.703} C_VEL
LIN {X 0,Y 425.365,Z 327.811,A -85,B 0,C 180,E1 -9703.687,E2 -9703.687} C_VEL
LIN {X 0,Y 425.41,Z 327.805,A -85,B 0,C 180,E1 -9707.598,E2 -9707.598} C_VEL
LIN {X 0,Y 425.42,Z 327.799,A -85,B 0,C 180,E1 -9711.449,E2 -9711.449} C_VEL
LIN {X 0,Y 425.531,Z 327.787,A -85,B 0,C 180,E1 -9714.313,E2 -9714.313} C_VEL
LIN {X 0,Y 425.547,Z 327.788,A -85,B 0,C 180,E1 -9718.107,E2 -9718.107} C_VEL
LIN {X 0,Y 425.676,Z 327.769,A -85,B 0,C 180,E1 -9720,E2 -9720} C_VEL
LIN {X 0,Y 425.544,Z 327.79,A -85,B 0,C 180,E1 -9722.84,E2 -9722.84} C_VEL
LIN {X 0,Y 425.556,Z 327.79,A -85,B 0,C 180,E1 -9725.686,E2 -9725.686} C_VEL
LIN {X 0,Y 425.418,Z 327.804,A -85,B 0,C 180,E1 -9728.55,E2 -9728.55} C_VEL
LIN {X 0,Y 425.406,Z 327.808,A -85,B 0,C 180,E1 -9732.402,E2 -9732.402} C_VEL
LIN {X 0,Y 425.375,Z 327.813,A -85,B 0,C 180,E1 -9736.312,E2 -9736.312} C_VEL
LIN {X 0,Y 425.339,Z 327.818,A -85,B 0,C 180,E1 -9739.65,E2 -9739.65} C_VEL
LIN {X 0,Y 425.313,Z 327.818,A -85,B 0,C 180,E1 -9742.337,E2 -9742.337} C_VEL
LIN {X 0,Y 425.273,Z 327.824,A -85,B 0,C 180,E1 -9745.446,E2 -9745.446} C_VEL
LIN {X 0,Y 425.308,Z 327.821,A -85,B 0,C 180,E1 -9748.633,E2 -9748.633} C_VEL
LIN {X 0,Y 425.243,Z 327.829,A -85,B 0,C 180,E1 -9751.928,E2 -9751.928} C_VEL
LIN {X 0,Y 425.28,Z 327.825,A -85,B 0,C 180,E1 -9755.337,E2 -9755.337} C_VEL
LIN {X 0,Y 425.293,Z 327.821,A -85,B 0,C 180,E1 -9758.899,E2 -9758.899} C_VEL
LIN {X 0,Y 425.28,Z 327.884,A -85,B 0,C 180,E1 -9761.441,E2 -9761.441} C_VEL
LIN {X 0,Y 429.182,Z 340.727,A -85,B 0,C 180,E1 -9765.244,E2 -9765.244} C_VEL
LIN {X 0,Y 432.471,Z 351.716,A -85,B 0,C 180,E1 -9768.223,E2 -9768.223} C_VEL
LIN {X 0,Y 436.06,Z 364.495,A -85,B 0,C 180,E1 -9771.413,E2 -9771.413} C_VEL
LIN {X 0,Y 436.923,Z 368.421,A -85,B 0,C 180,E1 -9772.325,E2 -9772.325} C_VEL
LIN {X 0,Y 435.286,Z 381.021,A -85,B 0,C 180,E1 -9774.778,E2 -9774.778} C_VEL
LIN {X 0,Y 433.27,Z 397.83,A -85,B 0,C 180,E1 -9777.915,E2 -9777.915} C_VEL
LIN {X 0,Y 431.358,Z 416.477,A -85,B 0,C 180,E1 -9781.279,E2 -9781.279} C_VEL
LIN {X 0,Y 431.183,Z 418.406,A -85,B 0,C 180,E1 -9781.623,E2 -9781.623} C_VEL
LIN {X 0,Y 435.709,Z 441.585,A -85,B 0,C 180,E1 -9782.395,E2 -9782.395} C_VEL
LIN {X 0,Y 437.621,Z 452.232,A -85,B 0,C 180,E1 -9782.827,E2 -9782.827} C_VEL
LIN {X 0,Y 436.695,Z 468.209,A -85,B 0,C 180,E1 -9783.413,E2 -9783.413} C_VEL
LIN {X 0,Y 435.523,Z 483.958,A -85,B 0,C 180,E1 -9784.173,E2 -9784.173} C_VEL
LIN {X 0,Y 434.26,Z 499.39,A -85,B 0,C 180,E1 -9785.119,E2 -9785.119} C_VEL
LIN {X 0,Y 432.85,Z 513.706,A -85,B 0,C 180,E1 -9786.182,E2 -9786.182} C_VEL
LIN {X 0,Y 431.396,Z 528.368,A -85,B 0,C 180,E1 -9787.493,E2 -9787.493} C_VEL
LIN {X 0,Y 429.945,Z 541.846,A -85,B 0,C 180,E1 -9788.926,E2 -9788.926} C_VEL
LIN {X 0,Y 428.729,Z 553.363,A -85,B 0,C 180,E1 -9790.367,E2 -9790.367} C_VEL
LIN {X 0,Y 427.537,Z 564.799,A -85,B 0,C 180,E1 -9792.039,E2 -9792.039} C_VEL
LIN {X 0,Y 426.548,Z 576.029,A -85,B 0,C 180,E1 -9793.982,E2 -9793.982} C_VEL
LIN {X 0,Y 425.644,Z 585.369,A -85,B 0,C 180,E1 -9795.907,E2 -9795.907} C_VEL
LIN {X 0,Y 425.12,Z 592.297,A -85,B 0,C 180,E1 -9797.592,E2 -9797.592} C_VEL
LIN {X 0,Y 424.638,Z 598.87,A -85,B 0,C 180,E1 -9799.513,E2 -9799.513} C_VEL
LIN {X 0,Y 424.402,Z 604.262,A -85,B 0,C 180,E1 -9801.431,E2 -9801.431} C_VEL
LIN {X 0,Y 424.314,Z 608.444,A -85,B 0,C 180,E1 -9803.344,E2 -9803.344} C_VEL
LIN {X 0,Y 424.175,Z 611.539,A -85,B 0,C 180,E1 -9805.25,E2 -9805.25} C_VEL
LIN {X 0,Y 424.165,Z 613.577,A -85,B 0,C 180,E1 -9807.153,E2 -9807.153} C_VEL
LIN {X 0,Y 424.11,Z 614.575,A -85,B 0,C 180,E1 -9809.053,E2 -9809.053} C_VEL
LIN {X 0,Y 424.111,Z 614.565,A -85,B 0,C 180,E1 -9810.952,E2 -9810.952} C_VEL
LIN {X 0,Y 424.166,Z 613.528,A -85,B 0,C 180,E1 -9812.851,E2 -9812.851} C_VEL
LIN {X 0,Y 424.177,Z 611.458,A -85,B 0,C 180,E1 -9814.754,E2 -9814.754} C_VEL
LIN {X 0,Y 424.317,Z 608.31,A -85,B 0,C 180,E1 -9816.66,E2 -9816.66} C_VEL
LIN {X 0,Y 424.436,Z 604.063,A -85,B 0,C 180,E1 -9818.573,E2 -9818.573} C_VEL
LIN {X 0,Y 424.649,Z 598.578,A -85,B 0,C 180,E1 -9820.491,E2 -9820.491} C_VEL
LIN {X 0,Y 425.158,Z 591.883,A -85,B 0,C 180,E1 -9822.411,E2 -9822.411} C_VEL
LIN {X 0,Y 425.753,Z 583.733,A -85,B 0,C 180,E1 -9824.338,E2 -9824.338} C_VEL
LIN {X 0,Y 426.669,Z 573.962,A -85,B 0,C 180,E1 -9826.263,E2 -9826.263} C_VEL
LIN {X 0,Y 427.508,Z 563.932,A -85,B 0,C 180,E1 -9827.942,E2 -9827.942} C_VEL
LIN {X 0,Y 428.713,Z 552.048,A -85,B 0,C 180,E1 -9829.639,E2 -9829.639} C_VEL
LIN {X 0,Y 430.062,Z 538.834,A -85,B 0,C 180,E1 -9831.237,E2 -9831.237} C_VEL
LIN {X 0,Y 431.425,Z 525.11,A -85,B 0,C 180,E1 -9832.637,E2 -9832.637} C_VEL
LIN {X 0,Y 432.76,Z 511.195,A -85,B 0,C 180,E1 -9833.828,E2 -9833.828} C_VEL
LIN {X 0,Y 434.082,Z 496.309,A -85,B 0,C 180,E1 -9834.897,E2 -9834.897} C_VEL
LIN {X 0,Y 435.365,Z 480.193,A -85,B 0,C 180,E1 -9835.842,E2 -9835.842} C_VEL
LIN {X 0,Y 436.452,Z 464.084,A -85,B 0,C 180,E1 -9836.588,E2 -9836.588} C_VEL
LIN {X 0,Y 437.1,Z 450.832,A -85,B 0,C 180,E1 -9837.065,E2 -9837.065} C_VEL
LIN {X 0,Y 433.572,Z 433.264,A -85,B 0,C 180,E1 -9837.758,E2 -9837.758} C_VEL
LIN {X 0,Y 430.834,Z 417.013,A -85,B 0,C 180,E1 -9838.289,E2 -9838.289} C_VEL
LIN {X 0,Y 432.42,Z 400.098,A -85,B 0,C 180,E1 -9841.34,E2 -9841.34} C_VEL
LIN {X 0,Y 434.6,Z 384.15,A -85,B 0,C 180,E1 -9844.473,E2 -9844.473} C_VEL
LIN {X 0,Y 437.145,Z 371.001,A -85,B 0,C 180,E1 -9847.368,E2 -9847.368} C_VEL
LIN {X 0,Y 437.27,Z 368.415,A -85,B 0,C 180,E1 -9848.043,E2 -9848.043} C_VEL
LIN {X 0,Y 436.374,Z 364.24,A -85,B 0,C 180,E1 -9849.371,E2 -9849.371} C_VEL
LIN {X 0,Y 434.76,Z 358.765,A -85,B 0,C 180,E1 -9851.514,E2 -9851.514} C_VEL
LIN {X 0,Y 433.67,Z 355.45,A -85,B 0,C 180,E1 -9853.176,E2 -9853.176} C_VEL
LIN {X 0,Y 432.976,Z 353.462,A -85,B 0,C 180,E1 -9854.423,E2 -9854.423} C_VEL
LIN {X 0,Y 432.462,Z 351.908,A -85,B 0,C 180,E1 -9855.67,E2 -9855.67} C_VEL
LIN {X 0,Y 431.655,Z 350.08,A -85,B 0,C 180,E1 -9858.123,E2 -9858.123} C_VEL
LIN {X 0,Y 431.163,Z 349.775,A -85,B 0,C 180,E1 -9860.528,E2 -9860.528} C_VEL
LIN {X 0,Y 430.853,Z 350.659,A -85,B 0,C 180,E1 -9862.877,E2 -9862.877} C_VEL
LIN {X 0,Y 430.365,Z 352.539,A -85,B 0,C 180,E1 -9865.141,E2 -9865.141} C_VEL
LIN {X 0,Y 429.176,Z 356.413,A -85,B 0,C 180,E1 -9868.398,E2 -9868.398} C_VEL
LIN {X 0,Y 428.387,Z 360.799,A -85,B 0,C 180,E1 -9871.591,E2 -9871.591} C_VEL
LIN {X 0,Y 427.873,Z 365.408,A -85,B 0,C 180,E1 -9874.719,E2 -9874.719} C_VEL
LIN {X 0,Y 427.437,Z 370.216,A -85,B 0,C 180,E1 -9877.78,E2 -9877.78} C_VEL
LIN {X 0,Y 427.015,Z 375.925,A -85,B 0,C 180,E1 -9881.262,E2 -9881.262} C_VEL
LIN {X 0,Y 427.036,Z 376.195,A -85,B 0,C 180,E1 -9881.331,E2 -9881.331} C_VEL
LIN {X 0,Y 432.285,Z 390.22,A -85,B 0,C 180,E1 -9882.39,E2 -9882.39} C_VEL
LIN {X 0,Y 433.383,Z 394.294,A -85,B 0,C 180,E1 -9882.69,E2 -9882.69} C_VEL
LIN {X 0,Y 432.465,Z 408.516,A -85,B 0,C 180,E1 -9883.548,E2 -9883.548} C_VEL
LIN {X 0,Y 431.583,Z 420.249,A -85,B 0,C 180,E1 -9884.44,E2 -9884.44} C_VEL
LIN {X 0,Y 430.599,Z 432.537,A -85,B 0,C 180,E1 -9885.588,E2 -9885.588} C_VEL
LIN {X 0,Y 429.738,Z 442.841,A -85,B 0,C 180,E1 -9886.765,E2 -9886.765} C_VEL
LIN {X 0,Y 428.874,Z 452.88,A -85,B 0,C 180,E1 -9888.18,E2 -9888.18} C_VEL
LIN {X 0,Y 428.098,Z 461.118,A -85,B 0,C 180,E1 -9889.597,E2 -9889.597} C_VEL
LIN {X 0,Y 427.377,Z 468.577,A -85,B 0,C 180,E1 -9891.199,E2 -9891.199} C_VEL
LIN {X 0,Y 426.81,Z 473.185,A -85,B 0,C 180,E1 -9892.431,E2 -9892.431} C_VEL
LIN {X 0,Y 426.474,Z 477.346,A -85,B 0,C 180,E1 -9893.851,E2 -9893.851} C_VEL
LIN {X 0,Y 426.223,Z 480.468,A -85,B 0,C 180,E1 -9895.271,E2 -9895.271} C_VEL
LIN {X 0,Y 426.048,Z 482.03,A -85,B 0,C 180,E1 -9896.217,E2 -9896.217} C_VEL
LIN {X 0,Y 425.866,Z 483.139,A -85,B 0,C 180,E1 -9897.163,E2 -9897.163} C_VEL
LIN {X 0,Y 425.656,Z 483.853,A -85,B 0,C 180,E1 -9898.108,E2 -9898.108} C_VEL
LIN {X 0,Y 425.566,Z 484.154,A -85,B 0,C 180,E1 -9899.054,E2 -9899.054} C_VEL
LIN {X 0,Y 425.492,Z 484.057,A -85,B 0,C 180,E1 -9900,E2 -9900} C_VEL
LIN {X 0,Y 425.427,Z 483.541,A -85,B 0,C 180,E1 -9900.947,E2 -9900.947} C_VEL
LIN {X 0,Y 425.408,Z 482.599,A -85,B 0,C 180,E1 -9901.894,E2 -9901.894} C_VEL
LIN {X 0,Y 425.524,Z 481.242,A -85,B 0,C 180,E1 -9902.84,E2 -9902.84} C_VEL
LIN {X 0,Y 425.499,Z 478.449,A -85,B 0,C 180,E1 -9904.263,E2 -9904.263} C_VEL
LIN {X 0,Y 425.53,Z 474.651,A -85,B 0,C 180,E1 -9905.687,E2 -9905.687} C_VEL
LIN {X 0,Y 425.937,Z 469.725,A -85,B 0,C 180,E1 -9907.109,E2 -9907.109} C_VEL
LIN {X 0,Y 426.253,Z 462.479,A -85,B 0,C 180,E1 -9908.773,E2 -9908.773} C_VEL
LIN {X 0,Y 426.73,Z 454.688,A -85,B 0,C 180,E1 -9910.198,E2 -9910.198} C_VEL
LIN {X 0,Y 427.15,Z 445.151,A -85,B 0,C 180,E1 -9911.628,E2 -9911.628} C_VEL
LIN {X 0,Y 427.862,Z 434.444,A -85,B 0,C 180,E1 -9912.933,E2 -9912.933} C_VEL
LIN {X 0,Y 428.453,Z 422.405,A -85,B 0,C 180,E1 -9914.123,E2 -9914.123} C_VEL
LIN {X 0,Y 429.034,Z 410.161,A -85,B 0,C 180,E1 -9915.102,E2 -9915.102} C_VEL
LIN {X 0,Y 429.699,Z 397.445,A -85,B 0,C 180,E1 -9915.9,E2 -9915.9} C_VEL
LIN {X 0,Y 430.004,Z 387.823,A -85,B 0,C 180,E1 -9916.391,E2 -9916.391} C_VEL
LIN {X 0,Y 426.77,Z 373.964,A -85,B 0,C 180,E1 -9917.077,E2 -9917.077} C_VEL
LIN {X 0,Y 425.023,Z 366.995,A -85,B 0,C 180,E1 -9917.378,E2 -9917.378} C_VEL
LIN {X 0,Y 425.104,Z 361.335,A -85,B 0,C 180,E1 -9920.315,E2 -9920.315} C_VEL
LIN {X 0,Y 425.262,Z 355.516,A -85,B 0,C 180,E1 -9923.368,E2 -9923.368} C_VEL
LIN {X 0,Y 425.454,Z 348.951,A -85,B 0,C 180,E1 -9926.87,E2 -9926.87} C_VEL
LIN {X 0,Y 425.675,Z 342.74,A -85,B 0,C 180,E1 -9930.236,E2 -9930.236} C_VEL
LIN {X 0,Y 425.899,Z 336.702,A -85,B 0,C 180,E1 -9933.56,E2 -9933.56} C_VEL
LIN {X 0,Y 425.823,Z 331.586,A -85,B 0,C 180,E1 -9936.453,E2 -9936.453} C_VEL
LIN {X 0,Y 425.304,Z 327.825,A -85,B 0,C 180,E1 -9938.747,E2 -9938.747} C_VEL
LIN {X 0,Y 425.291,Z 327.823,A -85,B 0,C 180,E1 -9941.956,E2 -9941.956} C_VEL
LIN {X 0,Y 425.294,Z 327.822,A -85,B 0,C 180,E1 -9945.282,E2 -9945.282} C_VEL
LIN {X 0,Y 425.274,Z 327.825,A -85,B 0,C 180,E1 -9948.619,E2 -9948.619} C_VEL
LIN {X 0,Y 425.329,Z 327.947,A -85,B 0,C 180,E1 -9951.406,E2 -9951.406} C_VEL
LIN {X 0,Y 426.331,Z 333.643,A -85,B 0,C 180,E1 -9953.878,E2 -9953.878} C_VEL
LIN {X 0,Y 426.537,Z 338.297,A -85,B 0,C 180,E1 -9955.928,E2 -9955.928} C_VEL
LIN {X 0,Y 426.413,Z 345.642,A -85,B 0,C 180,E1 -9959.272,E2 -9959.272} C_VEL
LIN {X 0,Y 426.271,Z 353.295,A -85,B 0,C 180,E1 -9962.913,E2 -9962.913} C_VEL
LIN {X 0,Y 426.222,Z 361.295,A -85,B 0,C 180,E1 -9966.686,E2 -9966.686} C_VEL
LIN {X 0,Y 426.222,Z 368.862,A -85,B 0,C 180,E1 -9970.032,E2 -9970.032} C_VEL
LIN {X 0,Y 426.372,Z 376.597,A -85,B 0,C 180,E1 -9973.121,E2 -9973.121} C_VEL
LIN {X 0,Y 430.144,Z 388.968,A -85,B 0,C 180,E1 -9973.644,E2 -9973.644} C_VEL
LIN {X 0,Y 429.932,Z 401.411,A -85,B 0,C 180,E1 -9974.168,E2 -9974.168} C_VEL
LIN {X 0,Y 429.565,Z 413.381,A -85,B 0,C 180,E1 -9974.86,E2 -9974.86} C_VEL
LIN {X 0,Y 429.041,Z 425.293,A -85,B 0,C 180,E1 -9975.774,E2 -9975.774} C_VEL
LIN {X 0,Y 428.5,Z 436.234,A -85,B 0,C 180,E1 -9976.844,E2 -9976.844} C_VEL
LIN {X 0,Y 427.99,Z 445.07,A -85,B 0,C 180,E1 -9977.913,E2 -9977.913} C_VEL
LIN {X 0,Y 427.218,Z 454.578,A -85,B 0,C 180,E1 -9979.333,E2 -9979.333} C_VEL
LIN {X 0,Y 426.698,Z 462.19,A -85,B 0,C 180,E1 -9980.757,E2 -9980.757} C_VEL
LIN {X 0,Y 426.342,Z 467.952,A -85,B 0,C 180,E1 -9982.102,E2 -9982.102} C_VEL
LIN {X 0,Y 426.186,Z 470.229,A -85,B 0,C 180,E1 -9982.735,E2 -9982.735} C_VEL
LIN {X 0,Y 425.323,Z 472.727,A -85,B 0,C 180,E1 -9983.446,E2 -9983.446} C_VEL
LIN {X 0,Y 420.888,Z 477.775,A -85,B 0,C 180,E1 -9985.091,E2 -9985.091} C_VEL
LIN {X 0,Y 418.836,Z 479.998,A -85,B 0,C 180,E1 -9986.09,E2 -9986.09} C_VEL
LIN {X 0,Y 418.468,Z 480.822,A -85,B 0,C 180,E1 -9986.613,E2 -9986.613} C_VEL
LIN {X 0,Y 418.323,Z 482.514,A -85,B 0,C 180,E1 -9988.072,E2 -9988.072} C_VEL
LIN {X 0,Y 418.211,Z 483.355,A -85,B 0,C 180,E1 -9989.998,E2 -9989.998} C_VEL
LIN {X 0,Y 418.315,Z 482.593,A -85,B 0,C 180,E1 -9991.923,E2 -9991.923} C_VEL
LIN {X 0,Y 418.561,Z 480.313,A -85,B 0,C 180,E1 -9993.849,E2 -9993.849} C_VEL
LIN {X 0,Y 418.689,Z 477.529,A -85,B 0,C 180,E1 -9995.295,E2 -9995.295} C_VEL
LIN {X 0,Y 418.993,Z 473.724,A -85,B 0,C 180,E1 -9996.74,E2 -9996.74} C_VEL
LIN {X 0,Y 419.464,Z 468.124,A -85,B 0,C 180,E1 -9998.351,E2 -9998.351} C_VEL
LIN {X 0,Y 419.916,Z 461.387,A -85,B 0,C 180,E1 -9999.875,E2 -9999.875} C_VEL
LIN {X 0,Y 420.63,Z 453.345,A -85,B 0,C 180,E1 -10001.319,E2 -10001.319} C_VEL
LIN {X 0,Y 421.175,Z 445.064,A -85,B 0,C 180,E1 -10002.526,E2 -10002.526} C_VEL
LIN {X 0,Y 421.805,Z 434.865,A -85,B 0,C 180,E1 -10003.732,E2 -10003.732} C_VEL
LIN {X 0,Y 422.319,Z 425.818,A -85,B 0,C 180,E1 -10004.601,E2 -10004.601} C_VEL
LIN {X 0,Y 422.746,Z 415.322,A -85,B 0,C 180,E1 -10005.423,E2 -10005.423} C_VEL
LIN {X 0,Y 423.219,Z 403.208,A -85,B 0,C 180,E1 -10006.147,E2 -10006.147} C_VEL
LIN {X 0,Y 423.395,Z 390.596,A -85,B 0,C 180,E1 -10006.698,E2 -10006.698} C_VEL
LIN {X 0,Y 419.497,Z 377.603,A -85,B 0,C 180,E1 -10007.263,E2 -10007.263} C_VEL
LIN {X 0,Y 419.312,Z 369.272,A -85,B 0,C 180,E1 -10010.605,E2 -10010.605} C_VEL
LIN {X 0,Y 419.277,Z 362.219,A -85,B 0,C 180,E1 -10013.718,E2 -10013.718} C_VEL
LIN {X 0,Y 419.334,Z 354.558,A -85,B 0,C 180,E1 -10017.342,E2 -10017.342} C_VEL
LIN {X 0,Y 419.477,Z 347.359,A -85,B 0,C 180,E1 -10020.727,E2 -10020.727} C_VEL
LIN {X 0,Y 419.618,Z 339.998,A -85,B 0,C 180,E1 -10024.127,E2 -10024.127} C_VEL
LIN {X 0,Y 419.352,Z 334.751,A -85,B 0,C 180,E1 -10026.443,E2 -10026.443} C_VEL
LIN {X 0,Y 418.224,Z 328.704,A -85,B 0,C 180,E1 -10029.058,E2 -10029.058} C_VEL
LIN {X 0,Y 418.21,Z 328.705,A -85,B 0,C 180,E1 -10032.318,E2 -10032.318} C_VEL
LIN {X 0,Y 418.244,Z 328.702,A -85,B 0,C 180,E1 -10035.109,E2 -10035.109} C_VEL
LIN {X 0,Y 418.277,Z 328.693,A -85,B 0,C 180,E1 -10037.771,E2 -10037.771} C_VEL
LIN {X 0,Y 418.251,Z 328.698,A -85,B 0,C 180,E1 -10041.558,E2 -10041.558} C_VEL
LIN {X 0,Y 418.241,Z 328.699,A -85,B 0,C 180,E1 -10045.157,E2 -10045.157} C_VEL
LIN {X 0,Y 418.226,Z 328.701,A -85,B 0,C 180,E1 -10047.47,E2 -10047.47} C_VEL
LIN {X 0,Y 418.248,Z 328.698,A -85,B 0,C 180,E1 -10050.893,E2 -10050.893} C_VEL
LIN {X 0,Y 418.254,Z 328.693,A -85,B 0,C 180,E1 -10054.094,E2 -10054.094} C_VEL
LIN {X 0,Y 418.276,Z 328.689,A -85,B 0,C 180,E1 -10057.528,E2 -10057.528} C_VEL
LIN {X 0,Y 418.295,Z 328.689,A -85,B 0,C 180,E1 -10060.364,E2 -10060.364} C_VEL
LIN {X 0,Y 418.293,Z 328.694,A -85,B 0,C 180,E1 -10063.403,E2 -10063.403} C_VEL
LIN {X 0,Y 418.332,Z 328.688,A -85,B 0,C 180,E1 -10066.992,E2 -10066.992} C_VEL
LIN {X 0,Y 418.341,Z 328.68,A -85,B 0,C 180,E1 -10070.328,E2 -10070.328} C_VEL
LIN {X 0,Y 418.47,Z 328.672,A -85,B 0,C 180,E1 -10073.248,E2 -10073.248} C_VEL
LIN {X 0,Y 418.315,Z 328.684,A -85,B 0,C 180,E1 -10075.181,E2 -10075.181} C_VEL
LIN {X 0,Y 418.516,Z 328.664,A -85,B 0,C 180,E1 -10078.075,E2 -10078.075} C_VEL
LIN {X 0,Y 418.646,Z 328.644,A -85,B 0,C 180,E1 -10080,E2 -10080} C_VEL
LIN {X 0,Y 418.498,Z 328.667,A -85,B 0,C 180,E1 -10082.887,E2 -10082.887} C_VEL
LIN {X 0,Y 418.511,Z 328.669,A -85,B 0,C 180,E1 -10085.782,E2 -10085.782} C_VEL
LIN {X 0,Y 418.376,Z 328.682,A -85,B 0,C 180,E1 -10088.695,E2 -10088.695} C_VEL
LIN {X 0,Y 418.311,Z 328.691,A -85,B 0,C 180,E1 -10091.631,E2 -10091.631} C_VEL
LIN {X 0,Y 418.285,Z 328.696,A -85,B 0,C 180,E1 -10094.597,E2 -10094.597} C_VEL
LIN {X 0,Y 418.267,Z 328.697,A -85,B 0,C 180,E1 -10097.604,E2 -10097.604} C_VEL
LIN {X 0,Y 418.256,Z 328.697,A -85,B 0,C 180,E1 -10100.662,E2 -10100.662} C_VEL
LIN {X 0,Y 418.271,Z 328.696,A -85,B 0,C 180,E1 -10103.782,E2 -10103.782} C_VEL
LIN {X 0,Y 418.287,Z 328.694,A -85,B 0,C 180,E1 -10107.072,E2 -10107.072} C_VEL
LIN {X 0,Y 418.222,Z 328.703,A -85,B 0,C 180,E1 -10110.273,E2 -10110.273} C_VEL
LIN {X 0,Y 418.227,Z 328.704,A -85,B 0,C 180,E1 -10113.679,E2 -10113.679} C_VEL
LIN {X 0,Y 418.225,Z 328.703,A -85,B 0,C 180,E1 -10117.225,E2 -10117.225} C_VEL
LIN {X 0,Y 418.236,Z 328.796,A -85,B 0,C 180,E1 -10120.695,E2 -10120.695} C_VEL
LIN {X 0,Y 421.015,Z 338.207,A -85,B 0,C 180,E1 -10123.584,E2 -10123.584} C_VEL
LIN {X 0,Y 424.464,Z 349.28,A -85,B 0,C 180,E1 -10126.762,E2 -10126.762} C_VEL
LIN {X 0,Y 427.629,Z 360.425,A -85,B 0,C 180,E1 -10129.696,E2 -10129.696} C_VEL
LIN {X 0,Y 430.026,Z 369.497,A -85,B 0,C 180,E1 -10131.922,E2 -10131.922} C_VEL
LIN {X 0,Y 430.122,Z 372.241,A -85,B 0,C 180,E1 -10132.512,E2 -10132.512} C_VEL
LIN {X 0,Y 427.522,Z 390.265,A -85,B 0,C 180,E1 -10136.022,E2 -10136.022} C_VEL
LIN {X 0,Y 425.567,Z 407.24,A -85,B 0,C 180,E1 -10139.21,E2 -10139.21} C_VEL
LIN {X 0,Y 424.446,Z 418.238,A -85,B 0,C 180,E1 -10141.208,E2 -10141.208} C_VEL
LIN {X 0,Y 428.994,Z 442.106,A -85,B 0,C 180,E1 -10142.02,E2 -10142.02} C_VEL
LIN {X 0,Y 431.056,Z 453.2,A -85,B 0,C 180,E1 -10142.496,E2 -10142.496} C_VEL
LIN {X 0,Y 430.064,Z 469.033,A -85,B 0,C 180,E1 -10143.101,E2 -10143.101} C_VEL
LIN {X 0,Y 428.731,Z 485.513,A -85,B 0,C 180,E1 -10143.93,E2 -10143.93} C_VEL
LIN {X 0,Y 427.35,Z 501.429,A -85,B 0,C 180,E1 -10144.949,E2 -10144.949} C_VEL
LIN {X 0,Y 425.771,Z 516.69,A -85,B 0,C 180,E1 -10146.149,E2 -10146.149} C_VEL
LIN {X 0,Y 424.3,Z 530.711,A -85,B 0,C 180,E1 -10147.481,E2 -10147.481} C_VEL
LIN {X 0,Y 422.924,Z 542.687,A -85,B 0,C 180,E1 -10148.815,E2 -10148.815} C_VEL
LIN {X 0,Y 421.503,Z 555.714,A -85,B 0,C 180,E1 -10150.523,E2 -10150.523} C_VEL
LIN {X 0,Y 420.326,Z 566.948,A -85,B 0,C 180,E1 -10152.261,E2 -10152.261} C_VEL
LIN {X 0,Y 419.303,Z 577.508,A -85,B 0,C 180,E1 -10154.198,E2 -10154.198} C_VEL
LIN {X 0,Y 418.426,Z 586.438,A -85,B 0,C 180,E1 -10156.155,E2 -10156.155} C_VEL
LIN {X 0,Y 417.963,Z 593.063,A -85,B 0,C 180,E1 -10157.869,E2 -10157.869} C_VEL
LIN {X 0,Y 417.5,Z 599.363,A -85,B 0,C 180,E1 -10159.822,E2 -10159.822} C_VEL
LIN {X 0,Y 417.322,Z 604.418,A -85,B 0,C 180,E1 -10161.773,E2 -10161.773} C_VEL
LIN {X 0,Y 417.219,Z 608.247,A -85,B 0,C 180,E1 -10163.638,E2 -10163.638} C_VEL
LIN {X 0,Y 417.122,Z 610.576,A -85,B 0,C 180,E1 -10165.17,E2 -10165.17} C_VEL
LIN {X 0,Y 417.134,Z 612.615,A -85,B 0,C 180,E1 -10167.105,E2 -10167.105} C_VEL
LIN {X 0,Y 417.076,Z 613.605,A -85,B 0,C 180,E1 -10169.037,E2 -10169.037} C_VEL
LIN {X 0,Y 417.079,Z 613.583,A -85,B 0,C 180,E1 -10170.968,E2 -10170.968} C_VEL
LIN {X 0,Y 417.135,Z 612.527,A -85,B 0,C 180,E1 -10172.9,E2 -10172.9} C_VEL
LIN {X 0,Y 417.142,Z 610.432,A -85,B 0,C 180,E1 -10174.835,E2 -10174.835} C_VEL
LIN {X 0,Y 417.277,Z 607.256,A -85,B 0,C 180,E1 -10176.773,E2 -10176.773} C_VEL
LIN {X 0,Y 417.368,Z 602.968,A -85,B 0,C 180,E1 -10178.719,E2 -10178.719} C_VEL
LIN {X 0,Y 417.621,Z 597.45,A -85,B 0,C 180,E1 -10180.67,E2 -10180.67} C_VEL
LIN {X 0,Y 418.134,Z 590.695,A -85,B 0,C 180,E1 -10182.623,E2 -10182.623} C_VEL
LIN {X 0,Y 418.743,Z 582.493,A -85,B 0,C 180,E1 -10184.583,E2 -10184.583} C_VEL
LIN {X 0,Y 419.637,Z 572.636,A -85,B 0,C 180,E1 -10186.544,E2 -10186.544} C_VEL
LIN {X 0,Y 420.594,Z 562.456,A -85,B 0,C 180,E1 -10188.26,E2 -10188.26} C_VEL
LIN {X 0,Y 421.842,Z 550.556,A -85,B 0,C 180,E1 -10189.972,E2 -10189.972} C_VEL
LIN {X 0,Y 423.117,Z 538.675,A -85,B 0,C 180,E1 -10191.435,E2 -10191.435} C_VEL
LIN {X 0,Y 424.558,Z 524.661,A -85,B 0,C 180,E1 -10192.895,E2 -10192.895} C_VEL
LIN {X 0,Y 425.947,Z 510.863,A -85,B 0,C 180,E1 -10194.104,E2 -10194.104} C_VEL
LIN {X 0,Y 427.38,Z 495.72,A -85,B 0,C 180,E1 -10195.215,E2 -10195.215} C_VEL
LIN {X 0,Y 428.659,Z 480.307,A -85,B 0,C 180,E1 -10196.146,E2 -10196.146} C_VEL
LIN {X 0,Y 429.829,Z 464.068,A -85,B 0,C 180,E1 -10196.925,E2 -10196.925} C_VEL
LIN {X 0,Y 430.477,Z 451.941,A -85,B 0,C 180,E1 -10197.38,E2 -10197.38} C_VEL
LIN {X 0,Y 427.037,Z 434.119,A -85,B 0,C 180,E1 -10198.129,E2 -10198.129} C_VEL
LIN {X 0,Y 424.045,Z 416.522,A -85,B 0,C 180,E1 -10198.729,E2 -10198.729} C_VEL
LIN {X 0,Y 425.665,Z 401.05,A -85,B 0,C 180,E1 -10201.617,E2 -10201.617} C_VEL
LIN {X 0,Y 427.676,Z 387.2,A -85,B 0,C 180,E1 -10204.409,E2 -10204.409} C_VEL
LIN {X 0,Y 430.454,Z 373.611,A -85,B 0,C 180,E1 -10207.46,E2 -10207.46} C_VEL
LIN {X 0,Y 430.728,Z 371.45,A -85,B 0,C 180,E1 -10208.023,E2 -10208.023} C_VEL
LIN {X 0,Y 429.733,Z 366.534,A -85,B 0,C 180,E1 -10209.631,E2 -10209.631} C_VEL
LIN {X 0,Y 428.244,Z 361.46,A -85,B 0,C 180,E1 -10211.694,E2 -10211.694} C_VEL
LIN {X 0,Y 426.975,Z 357.609,A -85,B 0,C 180,E1 -10213.737,E2 -10213.737} C_VEL
LIN {X 0,Y 425.885,Z 354.545,A -85,B 0,C 180,E1 -10216.125,E2 -10216.125} C_VEL
LIN {X 0,Y 425.085,Z 352.952,A -85,B 0,C 180,E1 -10218.599,E2 -10218.599} C_VEL
LIN {X 0,Y 424.836,Z 352.669,A -85,B 0,C 180,E1 -10219.822,E2 -10219.822} C_VEL
LIN {X 0,Y 424.426,Z 353.116,A -85,B 0,C 180,E1 -10222.217,E2 -10222.217} C_VEL
LIN {X 0,Y 423.899,Z 354.623,A -85,B 0,C 180,E1 -10224.53,E2 -10224.53} C_VEL
LIN {X 0,Y 423.046,Z 356.875,A -85,B 0,C 180,E1 -10226.755,E2 -10226.755} C_VEL
LIN {X 0,Y 422.032,Z 360.87,A -85,B 0,C 180,E1 -10230.028,E2 -10230.028} C_VEL
LIN {X 0,Y 421.312,Z 365.327,A -85,B 0,C 180,E1 -10233.232,E2 -10233.232} C_VEL
LIN {X 0,Y 420.723,Z 370.57,A -85,B 0,C 180,E1 -10236.747,E2 -10236.747} C_VEL
LIN {X 0,Y 420.375,Z 374.77,A -85,B 0,C 180,E1 -10239.447,E2 -10239.447} C_VEL
LIN {X 0,Y 420.243,Z 377.148,A -85,B 0,C 180,E1 -10240.809,E2 -10240.809} C_VEL
LIN {X 0,Y 425.67,Z 391.505,A -85,B 0,C 180,E1 -10241.956,E2 -10241.956} C_VEL
LIN {X 0,Y 427.013,Z 396.129,A -85,B 0,C 180,E1 -10242.328,E2 -10242.328} C_VEL
LIN {X 0,Y 426.023,Z 410.02,A -85,B 0,C 180,E1 -10243.196,E2 -10243.196} C_VEL
LIN {X 0,Y 425.008,Z 422.741,A -85,B 0,C 180,E1 -10244.199,E2 -10244.199} C_VEL
LIN {X 0,Y 423.95,Z 434.663,A -85,B 0,C 180,E1 -10245.357,E2 -10245.357} C_VEL
LIN {X 0,Y 423.069,Z 444.719,A -85,B 0,C 180,E1 -10246.552,E2 -10246.552} C_VEL
LIN {X 0,Y 422.132,Z 454.648,A -85,B 0,C 180,E1 -10247.989,E2 -10247.989} C_VEL
LIN {X 0,Y 421.32,Z 462.754,A -85,B 0,C 180,E1 -10249.427,E2 -10249.427} C_VEL
LIN {X 0,Y 420.621,Z 469.349,A -85,B 0,C 180,E1 -10250.867,E2 -10250.867} C_VEL
LIN {X 0,Y 419.93,Z 474.676,A -85,B 0,C 180,E1 -10252.306,E2 -10252.306} C_VEL
LIN {X 0,Y 419.559,Z 478.789,A -85,B 0,C 180,E1 -10253.75,E2 -10253.75} C_VEL
LIN {X 0,Y 419.286,Z 481.844,A -85,B 0,C 180,E1 -10255.193,E2 -10255.193} C_VEL
LIN {X 0,Y 419.107,Z 483.36,A -85,B 0,C 180,E1 -10256.154,E2 -10256.154} C_VEL
LIN {X 0,Y 418.9,Z 484.434,A -85,B 0,C 180,E1 -10257.115,E2 -10257.115} C_VEL
LIN {X 0,Y 418.681,Z 485.119,A -85,B 0,C 180,E1 -10258.076,E2 -10258.076} C_VEL
LIN {X 0,Y 418.579,Z 485.391,A -85,B 0,C 180,E1 -10259.038,E2 -10259.038} C_VEL
LIN {X 0,Y 418.506,Z 485.266,A -85,B 0,C 180,E1 -10260,E2 -10260} C_VEL
LIN {X 0,Y 418.452,Z 484.708,A -85,B 0,C 180,E1 -10260.963,E2 -10260.963} C_VEL
LIN {X 0,Y 418.406,Z 483.741,A -85,B 0,C 180,E1 -10261.926,E2 -10261.926} C_VEL
LIN {X 0,Y 418.523,Z 482.349,A -85,B 0,C 180,E1 -10262.888,E2 -10262.888} C_VEL
LIN {X 0,Y 418.493,Z 479.493,A -85,B 0,C 180,E1 -10264.334,E2 -10264.334} C_VEL
LIN {X 0,Y 418.54,Z 475.628,A -85,B 0,C 180,E1 -10265.783,E2 -10265.783} C_VEL
LIN {X 0,Y 418.966,Z 470.634,A -85,B 0,C 180,E1 -10267.228,E2 -10267.228} C_VEL
LIN {X 0,Y 419.308,Z 463.323,A -85,B 0,C 180,E1 -10268.919,E2 -10268.919} C_VEL
LIN {X 0,Y 419.801,Z 455.453,A -85,B 0,C 180,E1 -10270.368,E2 -10270.368} C_VEL
LIN {X 0,Y 420.225,Z 445.832,A -85,B 0,C 180,E1 -10271.822,E2 -10271.822} C_VEL
LIN {X 0,Y 420.972,Z 435.051,A -85,B 0,C 180,E1 -10273.148,E2 -10273.148} C_VEL
LIN {X 0,Y 421.585,Z 422.929,A -85,B 0,C 180,E1 -10274.358,E2 -10274.358} C_VEL
LIN {X 0,Y 422.195,Z 410.693,A -85,B 0,C 180,E1 -10275.347,E2 -10275.347} C_VEL
LIN {X 0,Y 422.879,Z 397.85,A -85,B 0,C 180,E1 -10276.164,E2 -10276.164} C_VEL
LIN {X 0,Y 423.18,Z 388.966,A -85,B 0,C 180,E1 -10276.626,E2 -10276.626} C_VEL
LIN {X 0,Y 419.997,Z 375.331,A -85,B 0,C 180,E1 -10277.329,E2 -10277.329} C_VEL
LIN {X 0,Y 417.979,Z 367.383,A -85,B 0,C 180,E1 -10277.681,E2 -10277.681} C_VEL
LIN {X 0,Y 418.102,Z 361.649,A -85,B 0,C 180,E1 -10280.671,E2 -10280.671} C_VEL
LIN {X 0,Y 418.255,Z 355.785,A -85,B 0,C 180,E1 -10283.784,E2 -10283.784} C_VEL
LIN {X 0,Y 418.443,Z 349.61,A -85,B 0,C 180,E1 -10287.103,E2 -10287.103} C_VEL
LIN {X 0,Y 418.672,Z 343.868,A -85,B 0,C 180,E1 -10290.238,E2 -10290.238} C_VEL
LIN {X 0,Y 418.917,Z 337.785,A -85,B 0,C 180,E1 -10293.617,E2 -10293.617} C_VEL
LIN {X 0,Y 418.869,Z 332.982,A -85,B 0,C 180,E1 -10296.352,E2 -10296.352} C_VEL
LIN {X 0,Y 418.274,Z 328.701,A -85,B 0,C 180,E1 -10298.902,E2 -10298.902} C_VEL
LIN {X 0,Y 418.233,Z 328.702,A -85,B 0,C 180,E1 -10302.319,E2 -10302.319} C_VEL
LIN {X 0,Y 418.245,Z 328.699,A -85,B 0,C 180,E1 -10305.108,E2 -10305.108} C_VEL
LIN {X 0,Y 418.243,Z 328.702,A -85,B 0,C 180,E1 -10307.765,E2 -10307.765} C_VEL
LIN {X 0,Y 418.271,Z 328.813,A -85,B 0,C 180,E1 -10311.096,E2 -10311.096} C_VEL
LIN {X 0,Y 419.47,Z 335.689,A -85,B 0,C 180,E1 -10314.096,E2 -10314.096} C_VEL
LIN {X 0,Y 419.564,Z 341.019,A -85,B 0,C 180,E1 -10316.441,E2 -10316.441} C_VEL
LIN {X 0,Y 419.469,Z 347.11,A -85,B 0,C 180,E1 -10319.267,E2 -10319.267} C_VEL
LIN {X 0,Y 419.324,Z 354.27,A -85,B 0,C 180,E1 -10322.661,E2 -10322.661} C_VEL
LIN {X 0,Y 419.268,Z 361.979,A -85,B 0,C 180,E1 -10326.276,E2 -10326.276} C_VEL
LIN {X 0,Y 419.32,Z 368.995,A -85,B 0,C 180,E1 -10329.39,E2 -10329.39} C_VEL
LIN {X 0,Y 419.486,Z 377.617,A -85,B 0,C 180,E1 -10332.848,E2 -10332.848} C_VEL
LIN {X 0,Y 423.42,Z 390.953,A -85,B 0,C 180,E1 -10333.412,E2 -10333.412} C_VEL
LIN {X 0,Y 423.135,Z 403.681,A -85,B 0,C 180,E1 -10333.969,E2 -10333.969} C_VEL
LIN {X 0,Y 422.786,Z 415.142,A -85,B 0,C 180,E1 -10334.661,E2 -10334.661} C_VEL
LIN {X 0,Y 422.243,Z 426.36,A -85,B 0,C 180,E1 -10335.54,E2 -10335.54} C_VEL
LIN {X 0,Y 421.668,Z 437.305,A -85,B 0,C 180,E1 -10336.627,E2 -10336.627} C_VEL
LIN {X 0,Y 421.132,Z 446.143,A -85,B 0,C 180,E1 -10337.713,E2 -10337.713} C_VEL
LIN {X 0,Y 420.324,Z 455.652,A -85,B 0,C 180,E1 -10339.156,E2 -10339.156} C_VEL
LIN {X 0,Y 419.801,Z 463.262,A -85,B 0,C 180,E1 -10340.604,E2 -10340.604} C_VEL
LIN {X 0,Y 419.406,Z 468.96,A -85,B 0,C 180,E1 -10341.953,E2 -10341.953} C_VEL
LIN {X 0,Y 419.012,Z 473.414,A -85,B 0,C 180,E1 -10343.255,E2 -10343.255} C_VEL
LIN {X 0,Y 418.693,Z 477.297,A -85,B 0,C 180,E1 -10344.701,E2 -10344.701} C_VEL
LIN {X 0,Y 418.468,Z 480.822,A -85,B 0,C 180,E1 -10346.613,E2 -10346.613} C_VEL
LIN {X 0,Y 417.72,Z 481.988,A -85,B 0,C 180,E1 -10347.401,E2 -10347.401} C_VEL
LIN {X 0,Y 414.747,Z 483.499,A -85,B 0,C 180,E1 -10348.687,E2 -10348.687} C_VEL
LIN {X 0,Y 412.295,Z 484.221,A -85,B 0,C 180,E1 -10349.731,E2 -10349.731} C_VEL
LIN {X 0,Y 411.277,Z 484.35,A -85,B 0,C 180,E1 -10350.542,E2 -10350.542} C_VEL
LIN {X 0,Y 411.212,Z 484.275,A -85,B 0,C 180,E1 -10350.817,E2 -10350.817} C_VEL
LIN {X 0,Y 411.309,Z 483.668,A -85,B 0,C 180,E1 -10351.956,E2 -10351.956} C_VEL
LIN {X 0,Y 411.45,Z 482.717,A -85,B 0,C 180,E1 -10352.935,E2 -10352.935} C_VEL
LIN {X 0,Y 411.558,Z 481.389,A -85,B 0,C 180,E1 -10353.914,E2 -10353.914} C_VEL
LIN {X 0,Y 411.699,Z 478.605,A -85,B 0,C 180,E1 -10355.385,E2 -10355.385} C_VEL
LIN {X 0,Y 412.027,Z 474.798,A -85,B 0,C 180,E1 -10356.855,E2 -10356.855} C_VEL
LIN {X 0,Y 412.54,Z 469.093,A -85,B 0,C 180,E1 -10358.519,E2 -10358.519} C_VEL
LIN {X 0,Y 413.001,Z 462.458,A -85,B 0,C 180,E1 -10360.042,E2 -10360.042} C_VEL
LIN {X 0,Y 413.754,Z 454.413,A -85,B 0,C 180,E1 -10361.51,E2 -10361.51} C_VEL
LIN {X 0,Y 414.325,Z 446.129,A -85,B 0,C 180,E1 -10362.736,E2 -10362.736} C_VEL
LIN {X 0,Y 415.006,Z 435.924,A -85,B 0,C 180,E1 -10363.962,E2 -10363.962} C_VEL
LIN {X 0,Y 415.535,Z 426.863,A -85,B 0,C 180,E1 -10364.846,E2 -10364.846} C_VEL
LIN {X 0,Y 415.979,Z 416.372,A -85,B 0,C 180,E1 -10365.681,E2 -10365.681} C_VEL
LIN {X 0,Y 416.467,Z 404.243,A -85,B 0,C 180,E1 -10366.416,E2 -10366.416} C_VEL
LIN {X 0,Y 416.584,Z 391.705,A -85,B 0,C 180,E1 -10366.975,E2 -10366.975} C_VEL
LIN {X 0,Y 412.88,Z 379.783,A -85,B 0,C 180,E1 -10367.499,E2 -10367.499} C_VEL
LIN {X 0,Y 412.572,Z 378.613,A -85,B 0,C 180,E1 -10367.555,E2 -10367.555} C_VEL
LIN {X 0,Y 412.416,Z 371.419,A -85,B 0,C 180,E1 -10370.403,E2 -10370.403} C_VEL
LIN {X 0,Y 412.369,Z 364.094,A -85,B 0,C 180,E1 -10373.607,E2 -10373.607} C_VEL
LIN {X 0,Y 412.387,Z 355.975,A -85,B 0,C 180,E1 -10377.393,E2 -10377.393} C_VEL
LIN {X 0,Y 412.553,Z 348.898,A -85,B 0,C 180,E1 -10380.731,E2 -10380.731} C_VEL
LIN {X 0,Y 412.686,Z 341.411,A -85,B 0,C 180,E1 -10384.19,E2 -10384.19} C_VEL
LIN {X 0,Y 412.569,Z 337.375,A -85,B 0,C 180,E1 -10385.99,E2 -10385.99} C_VEL
LIN {X 0,Y 411.529,Z 331.288,A -85,B 0,C 180,E1 -10388.666,E2 -10388.666} C_VEL
LIN {X 0,Y 411.185,Z 329.582,A -85,B 0,C 180,E1 -10389.474,E2 -10389.474} C_VEL
LIN {X 0,Y 411.157,Z 329.583,A -85,B 0,C 180,E1 -10393.131,E2 -10393.131} C_VEL
LIN {X 0,Y 411.213,Z 329.574,A -85,B 0,C 180,E1 -10395.87,E2 -10395.87} C_VEL
LIN {X 0,Y 411.195,Z 329.58,A -85,B 0,C 180,E1 -10398.762,E2 -10398.762} C_VEL
LIN {X 0,Y 411.189,Z 329.577,A -85,B 0,C 180,E1 -10402.025,E2 -10402.025} C_VEL
LIN {X 0,Y 411.188,Z 329.582,A -85,B 0,C 180,E1 -10405.664,E2 -10405.664} C_VEL
LIN {X 0,Y 411.169,Z 329.581,A -85,B 0,C 180,E1 -10409.15,E2 -10409.15} C_VEL
LIN {X 0,Y 411.238,Z 329.572,A -85,B 0,C 180,E1 -10412.52,E2 -10412.52} C_VEL
LIN {X 0,Y 411.211,Z 329.576,A -85,B 0,C 180,E1 -10415.783,E2 -10415.783} C_VEL
LIN {X 0,Y 411.221,Z 329.573,A -85,B 0,C 180,E1 -10418.967,E2 -10418.967} C_VEL
LIN {X 0,Y 411.23,Z 329.569,A -85,B 0,C 180,E1 -10422.084,E2 -10422.084} C_VEL
LIN {X 0,Y 411.24,Z 329.564,A -85,B 0,C 180,E1 -10425.146,E2 -10425.146} C_VEL
LIN {X 0,Y 411.283,Z 329.568,A -85,B 0,C 180,E1 -10428.167,E2 -10428.167} C_VEL
LIN {X 0,Y 411.457,Z 329.546,A -85,B 0,C 180,E1 -10432.146,E2 -10432.146} C_VEL
LIN {X 0,Y 411.452,Z 329.542,A -85,B 0,C 180,E1 -10434.117,E2 -10434.117} C_VEL
LIN {X 0,Y 411.485,Z 329.54,A -85,B 0,C 180,E1 -10438.042,E2 -10438.042} C_VEL
LIN {X 0,Y 411.615,Z 329.52,A -85,B 0,C 180,E1 -10440,E2 -10440} C_VEL
LIN {X 0,Y 411.453,Z 329.544,A -85,B 0,C 180,E1 -10442.937,E2 -10442.937} C_VEL
LIN {X 0,Y 411.47,Z 329.546,A -85,B 0,C 180,E1 -10445.882,E2 -10445.882} C_VEL
LIN {X 0,Y 411.457,Z 329.547,A -85,B 0,C 180,E1 -10447.853,E2 -10447.853} C_VEL
LIN {X 0,Y 411.277,Z 329.567,A -85,B 0,C 180,E1 -10451.833,E2 -10451.833} C_VEL
LIN {X 0,Y 411.242,Z 329.572,A -85,B 0,C 180,E1 -10454.853,E2 -10454.853} C_VEL
LIN {X 0,Y 411.232,Z 329.576,A -85,B 0,C 180,E1 -10457.916,E2 -10457.916} C_VEL
LIN {X 0,Y 411.219,Z 329.574,A -85,B 0,C 180,E1 -10461.032,E2 -10461.032} C_VEL
LIN {X 0,Y 411.207,Z 329.575,A -85,B 0,C 180,E1 -10464.216,E2 -10464.216} C_VEL
LIN {X 0,Y 411.236,Z 329.57,A -85,B 0,C 180,E1 -10467.479,E2 -10467.479} C_VEL
LIN {X 0,Y 411.167,Z 329.582,A -85,B 0,C 180,E1 -10470.849,E2 -10470.849} C_VEL
LIN {X 0,Y 411.185,Z 329.579,A -85,B 0,C 180,E1 -10474.335,E2 -10474.335} C_VEL
LIN {X 0,Y 411.18,Z 329.578,A -85,B 0,C 180,E1 -10477.975,E2 -10477.975} C_VEL
LIN {X 0,Y 411.194,Z 329.647,A -85,B 0,C 180,E1 -10479.914,E2 -10479.914} C_VEL
LIN {X 0,Y 414.221,Z 339.937,A -85,B 0,C 180,E1 -10483.154,E2 -10483.154} C_VEL
LIN {X 0,Y 417.635,Z 350.933,A -85,B 0,C 180,E1 -10486.378,E2 -10486.378} C_VEL
LIN {X 0,Y 420.77,Z 362.019,A -85,B 0,C 180,E1 -10489.356,E2 -10489.356} C_VEL
LIN {X 0,Y 423.412,Z 372.038,A -85,B 0,C 180,E1 -10491.86,E2 -10491.86} C_VEL
LIN {X 0,Y 423.39,Z 374.369,A -85,B 0,C 180,E1 -10492.364,E2 -10492.364} C_VEL
LIN {X 0,Y 420.858,Z 391.199,A -85,B 0,C 180,E1 -10495.699,E2 -10495.699} C_VEL
LIN {X 0,Y 418.772,Z 408.253,A -85,B 0,C 180,E1 -10498.975,E2 -10498.975} C_VEL
LIN {X 0,Y 417.698,Z 418.089,A -85,B 0,C 180,E1 -10500.776,E2 -10500.776} C_VEL
LIN {X 0,Y 422.287,Z 442.453,A -85,B 0,C 180,E1 -10501.629,E2 -10501.629} C_VEL
LIN {X 0,Y 424.47,Z 454.145,A -85,B 0,C 180,E1 -10502.152,E2 -10502.152} C_VEL
LIN {X 0,Y 423.428,Z 469.794,A -85,B 0,C 180,E1 -10502.779,E2 -10502.779} C_VEL
LIN {X 0,Y 422.156,Z 484.956,A -85,B 0,C 180,E1 -10503.559,E2 -10503.559} C_VEL
LIN {X 0,Y 420.682,Z 501.027,A -85,B 0,C 180,E1 -10504.606,E2 -10504.606} C_VEL
LIN {X 0,Y 419.122,Z 515.339,A -85,B 0,C 180,E1 -10505.746,E2 -10505.746} C_VEL
LIN {X 0,Y 417.57,Z 529.456,A -85,B 0,C 180,E1 -10507.098,E2 -10507.098} C_VEL
LIN {X 0,Y 416.161,Z 541.511,A -85,B 0,C 180,E1 -10508.453,E2 -10508.453} C_VEL
LIN {X 0,Y 414.848,Z 552.892,A -85,B 0,C 180,E1 -10509.94,E2 -10509.94} C_VEL
LIN {X 0,Y 413.57,Z 564.207,A -85,B 0,C 180,E1 -10511.68,E2 -10511.68} C_VEL
LIN {X 0,Y 412.585,Z 573.913,A -85,B 0,C 180,E1 -10513.425,E2 -10513.425} C_VEL
LIN {X 0,Y 411.619,Z 583.323,A -85,B 0,C 180,E1 -10515.416,E2 -10515.416} C_VEL
LIN {X 0,Y 411.076,Z 590.276,A -85,B 0,C 180,E1 -10517.161,E2 -10517.161} C_VEL
LIN {X 0,Y 410.586,Z 596.904,A -85,B 0,C 180,E1 -10519.15,E2 -10519.15} C_VEL
LIN {X 0,Y 410.295,Z 602.318,A -85,B 0,C 180,E1 -10521.134,E2 -10521.134} C_VEL
LIN {X 0,Y 410.217,Z 606.509,A -85,B 0,C 180,E1 -10523.115,E2 -10523.115} C_VEL
LIN {X 0,Y 410.071,Z 609.614,A -85,B 0,C 180,E1 -10525.087,E2 -10525.087} C_VEL
LIN {X 0,Y 410.103,Z 611.648,A -85,B 0,C 180,E1 -10527.055,E2 -10527.055} C_VEL
LIN {X 0,Y 410.042,Z 612.635,A -85,B 0,C 180,E1 -10529.02,E2 -10529.02} C_VEL
LIN {X 0,Y 410.047,Z 612.597,A -85,B 0,C 180,E1 -10530.984,E2 -10530.984} C_VEL
LIN {X 0,Y 410.105,Z 611.527,A -85,B 0,C 180,E1 -10532.949,E2 -10532.949} C_VEL
LIN {X 0,Y 410.108,Z 609.405,A -85,B 0,C 180,E1 -10534.918,E2 -10534.918} C_VEL
LIN {X 0,Y 410.223,Z 606.2,A -85,B 0,C 180,E1 -10536.89,E2 -10536.89} C_VEL
LIN {X 0,Y 410.315,Z 601.876,A -85,B 0,C 180,E1 -10538.87,E2 -10538.87} C_VEL
LIN {X 0,Y 410.6,Z 596.313,A -85,B 0,C 180,E1 -10540.855,E2 -10540.855} C_VEL
LIN {X 0,Y 411.157,Z 588.836,A -85,B 0,C 180,E1 -10543.016,E2 -10543.016} C_VEL
LIN {X 0,Y 411.837,Z 580.09,A -85,B 0,C 180,E1 -10545.086,E2 -10545.086} C_VEL
LIN {X 0,Y 412.692,Z 571.325,A -85,B 0,C 180,E1 -10546.83,E2 -10546.83} C_VEL
LIN {X 0,Y 413.711,Z 561.061,A -85,B 0,C 180,E1 -10548.575,E2 -10548.575} C_VEL
LIN {X 0,Y 414.99,Z 549.063,A -85,B 0,C 180,E1 -10550.317,E2 -10550.317} C_VEL
LIN {X 0,Y 416.447,Z 535.984,A -85,B 0,C 180,E1 -10551.926,E2 -10551.926} C_VEL
LIN {X 0,Y 417.981,Z 521.724,A -85,B 0,C 180,E1 -10553.407,E2 -10553.407} C_VEL
LIN {X 0,Y 419.48,Z 507.667,A -85,B 0,C 180,E1 -10554.632,E2 -10554.632} C_VEL
LIN {X 0,Y 420.949,Z 492.511,A -85,B 0,C 180,E1 -10555.729,E2 -10555.729} C_VEL
LIN {X 0,Y 422.19,Z 478.35,A -85,B 0,C 180,E1 -10556.577,E2 -10556.577} C_VEL
LIN {X 0,Y 423.361,Z 462.131,A -85,B 0,C 180,E1 -10557.36,E2 -10557.36} C_VEL
LIN {X 0,Y 423.871,Z 453.086,A -85,B 0,C 180,E1 -10557.714,E2 -10557.714} C_VEL
LIN {X 0,Y 420.635,Z 435.411,A -85,B 0,C 180,E1 -10558.506,E2 -10558.506} C_VEL
LIN {X 0,Y 417.801,Z 418.517,A -85,B 0,C 180,E1 -10559.109,E2 -10559.109} C_VEL
LIN {X 0,Y 417.345,Z 415.892,A -85,B 0,C 180,E1 -10559.234,E2 -10559.234} C_VEL
LIN {X 0,Y 419.12,Z 400.699,A -85,B 0,C 180,E1 -10562.17,E2 -10562.17} C_VEL
LIN {X 0,Y 421.361,Z 387.045,A -85,B 0,C 180,E1 -10565.042,E2 -10565.042} C_VEL
LIN {X 0,Y 424.023,Z 375.139,A -85,B 0,C 180,E1 -10567.827,E2 -10567.827} C_VEL
LIN {X 0,Y 424.14,Z 373.461,A -85,B 0,C 180,E1 -10568.294,E2 -10568.294} C_VEL
LIN {X 0,Y 423.311,Z 369.598,A -85,B 0,C 180,E1 -10569.611,E2 -10569.611} C_VEL
LIN {X 0,Y 421.769,Z 364.31,A -85,B 0,C 180,E1 -10571.801,E2 -10571.801} C_VEL
LIN {X 0,Y 420.909,Z 361.621,A -85,B 0,C 180,E1 -10573.205,E2 -10573.205} C_VEL
LIN {X 0,Y 419.806,Z 358.519,A -85,B 0,C 180,E1 -10575.322,E2 -10575.322} C_VEL
LIN {X 0,Y 418.968,Z 356.482,A -85,B 0,C 180,E1 -10577.57,E2 -10577.57} C_VEL
LIN {X 0,Y 418.541,Z 355.803,A -85,B 0,C 180,E1 -10579.09,E2 -10579.09} C_VEL
LIN {X 0,Y 418.018,Z 355.767,A -85,B 0,C 180,E1 -10581.533,E2 -10581.533} C_VEL
LIN {X 0,Y 417.482,Z 356.863,A -85,B 0,C 180,E1 -10583.908,E2 -10583.908} C_VEL
LIN {X 0,Y 416.646,Z 358.804,A -85,B 0,C 180,E1 -10586.176,E2 -10586.176} C_VEL
LIN {X 0,Y 415.383,Z 362.736,A -85,B 0,C 180,E1 -10589.644,E2 -10589.644} C_VEL
LIN {X 0,Y 414.607,Z 366.858,A -85,B 0,C 180,E1 -10592.763,E2 -10592.763} C_VEL
LIN {X 0,Y 413.964,Z 372.166,A -85,B 0,C 180,E1 -10596.462,E2 -10596.462} C_VEL
LIN {X 0,Y 413.418,Z 377.908,A -85,B 0,C 180,E1 -10600.194,E2 -10600.194} C_VEL
LIN {X 0,Y 413.674,Z 378.889,A -85,B 0,C 180,E1 -10600.308,E2 -10600.308} C_VEL
LIN {X 0,Y 418.674,Z 391.666,A -85,B 0,C 180,E1 -10601.402,E2 -10601.402} C_VEL
LIN {X 0,Y 420.622,Z 397.756,A -85,B 0,C 180,E1 -10601.929,E2 -10601.929} C_VEL
LIN {X 0,Y 419.628,Z 411.741,A -85,B 0,C 180,E1 -10602.837,E2 -10602.837} C_VEL
LIN {X 0,Y 418.474,Z 424.846,A -85,B 0,C 180,E1 -10603.913,E2 -10603.913} C_VEL
LIN {X 0,Y 417.32,Z 436.851,A -85,B 0,C 180,E1 -10605.119,E2 -10605.119} C_VEL
LIN {X 0,Y 416.237,Z 448.438,A -85,B 0,C 180,E1 -10606.576,E2 -10606.576} C_VEL
LIN {X 0,Y 415.286,Z 457.881,A -85,B 0,C 180,E1 -10608.036,E2 -10608.036} C_VEL
LIN {X 0,Y 414.437,Z 465.595,A -85,B 0,C 180,E1 -10609.496,E2 -10609.496} C_VEL
LIN {X 0,Y 413.533,Z 472.801,A -85,B 0,C 180,E1 -10611.202,E2 -10611.202} C_VEL
LIN {X 0,Y 413,Z 477.599,A -85,B 0,C 180,E1 -10612.668,E2 -10612.668} C_VEL
LIN {X 0,Y 412.495,Z 481.33,A -85,B 0,C 180,E1 -10614.133,E2 -10614.133} C_VEL
LIN {X 0,Y 412.37,Z 483.232,A -85,B 0,C 180,E1 -10615.112,E2 -10615.112} C_VEL
LIN {X 0,Y 412.158,Z 484.712,A -85,B 0,C 180,E1 -10616.089,E2 -10616.089} C_VEL
LIN {X 0,Y 411.953,Z 485.75,A -85,B 0,C 180,E1 -10617.067,E2 -10617.067} C_VEL
LIN {X 0,Y 411.723,Z 486.399,A -85,B 0,C 180,E1 -10618.044,E2 -10618.044} C_VEL
LIN {X 0,Y 411.611,Z 486.636,A -85,B 0,C 180,E1 -10619.022,E2 -10619.022} C_VEL
LIN {X 0,Y 411.516,Z 486.474,A -85,B 0,C 180,E1 -10620,E2 -10620} C_VEL
LIN {X 0,Y 411.471,Z 485.873,A -85,B 0,C 180,E1 -10620.979,E2 -10620.979} C_VEL
LIN {X 0,Y 411.401,Z 484.87,A -85,B 0,C 180,E1 -10621.958,E2 -10621.958} C_VEL
LIN {X 0,Y 411.521,Z 483.438,A -85,B 0,C 180,E1 -10622.937,E2 -10622.937} C_VEL
LIN {X 0,Y 411.488,Z 480.525,A -85,B 0,C 180,E1 -10624.408,E2 -10624.408} C_VEL
LIN {X 0,Y 411.551,Z 476.597,A -85,B 0,C 180,E1 -10625.881,E2 -10625.881} C_VEL
LIN {X 0,Y 411.997,Z 471.533,A -85,B 0,C 180,E1 -10627.351,E2 -10627.351} C_VEL
LIN {X 0,Y 412.367,Z 464.118,A -85,B 0,C 180,E1 -10629.071,E2 -10629.071} C_VEL
LIN {X 0,Y 412.849,Z 456.166,A -85,B 0,C 180,E1 -10630.545,E2 -10630.545} C_VEL
LIN {X 0,Y 413.312,Z 446.473,A -85,B 0,C 180,E1 -10632.023,E2 -10632.023} C_VEL
LIN {X 0,Y 414.056,Z 436.676,A -85,B 0,C 180,E1 -10633.247,E2 -10633.247} C_VEL
LIN {X 0,Y 414.707,Z 424.75,A -85,B 0,C 180,E1 -10634.476,E2 -10634.476} C_VEL
LIN {X 0,Y 415.306,Z 412.514,A -85,B 0,C 180,E1 -10635.5,E2 -10635.5} C_VEL
LIN {X 0,Y 416.061,Z 399.321,A -85,B 0,C 180,E1 -10636.373,E2 -10636.373} C_VEL
LIN {X 0,Y 416.336,Z 389.994,A -85,B 0,C 180,E1 -10636.874,E2 -10636.874} C_VEL
LIN {X 0,Y 412.973,Z 375.657,A -85,B 0,C 180,E1 -10637.63,E2 -10637.63} C_VEL
LIN {X 0,Y 410.944,Z 367.75,A -85,B 0,C 180,E1 -10637.994,E2 -10637.994} C_VEL
LIN {X 0,Y 411.083,Z 361.975,A -85,B 0,C 180,E1 -10641.041,E2 -10641.041} C_VEL
LIN {X 0,Y 411.243,Z 356.025,A -85,B 0,C 180,E1 -10644.215,E2 -10644.215} C_VEL
LIN {X 0,Y 411.468,Z 350.042,A -85,B 0,C 180,E1 -10647.463,E2 -10647.463} C_VEL
LIN {X 0,Y 411.706,Z 344.005,A -85,B 0,C 180,E1 -10650.805,E2 -10650.805} C_VEL
LIN {X 0,Y 411.917,Z 337.838,A -85,B 0,C 180,E1 -10654.266,E2 -10654.266} C_VEL
LIN {X 0,Y 411.799,Z 333.673,A -85,B 0,C 180,E1 -10656.679,E2 -10656.679} C_VEL
LIN {X 0,Y 411.21,Z 329.581,A -85,B 0,C 180,E1 -10659.225,E2 -10659.225} C_VEL
LIN {X 0,Y 411.187,Z 329.578,A -85,B 0,C 180,E1 -10662.694,E2 -10662.694} C_VEL
LIN {X 0,Y 411.176,Z 329.582,A -85,B 0,C 180,E1 -10665.88,E2 -10665.88} C_VEL
LIN {X 0,Y 411.167,Z 329.583,A -85,B 0,C 180,E1 -10668.772,E2 -10668.772} C_VEL
LIN {X 0,Y 411.232,Z 329.701,A -85,B 0,C 180,E1 -10670.775,E2 -10670.775} C_VEL
LIN {X 0,Y 412.316,Z 335.63,A -85,B 0,C 180,E1 -10673.373,E2 -10673.373} C_VEL
LIN {X 0,Y 412.682,Z 340.051,A -85,B 0,C 180,E1 -10675.319,E2 -10675.319} C_VEL
LIN {X 0,Y 412.567,Z 346.788,A -85,B 0,C 180,E1 -10678.402,E2 -10678.402} C_VEL
LIN {X 0,Y 412.417,Z 353.377,A -85,B 0,C 180,E1 -10681.499,E2 -10681.499} C_VEL
LIN {X 0,Y 412.306,Z 359.987,A -85,B 0,C 180,E1 -10684.612,E2 -10684.612} C_VEL
LIN {X 0,Y 412.367,Z 366.263,A -85,B 0,C 180,E1 -10687.478,E2 -10687.478} C_VEL
LIN {X 0,Y 412.439,Z 373.6,A -85,B 0,C 180,E1 -10690.591,E2 -10690.591} C_VEL
LIN {X 0,Y 412.563,Z 378.603,A -85,B 0,C 180,E1 -10692.548,E2 -10692.548} C_VEL
LIN {X 0,Y 416.695,Z 392.285,A -85,B 0,C 180,E1 -10693.148,E2 -10693.148} C_VEL
LIN {X 0,Y 416.39,Z 404.734,A -85,B 0,C 180,E1 -10693.702,E2 -10693.702} C_VEL
LIN {X 0,Y 416.013,Z 416.205,A -85,B 0,C 180,E1 -10694.405,E2 -10694.405} C_VEL
LIN {X 0,Y 415.455,Z 427.427,A -85,B 0,C 180,E1 -10695.299,E2 -10695.299} C_VEL
LIN {X 0,Y 414.843,Z 438.375,A -85,B 0,C 180,E1 -10696.403,E2 -10696.403} C_VEL
LIN {X 0,Y 414.304,Z 447.212,A -85,B 0,C 180,E1 -10697.507,E2 -10697.507} C_VEL
LIN {X 0,Y 413.435,Z 456.727,A -85,B 0,C 180,E1 -10698.973,E2 -10698.973} C_VEL
LIN {X 0,Y 412.882,Z 464.337,A -85,B 0,C 180,E1 -10700.445,E2 -10700.445} C_VEL
LIN {X 0,Y 412.476,Z 469.966,A -85,B 0,C 180,E1 -10701.799,E2 -10701.799} C_VEL
LIN {X 0,Y 412.046,Z 474.491,A -85,B 0,C 180,E1 -10703.141,E2 -10703.141} C_VEL
LIN {X 0,Y 411.707,Z 478.374,A -85,B 0,C 180,E1 -10704.61,E2 -10704.61} C_VEL
LIN {X 0,Y 411.471,Z 481.919,A -85,B 0,C 180,E1 -10706.57,E2 -10706.57} C_VEL
LIN {X 0,Y 411.315,Z 483.591,A -85,B 0,C 180,E1 -10708.039,E2 -10708.039} C_VEL
LIN {X 0,Y 411.194,Z 484.432,A -85,B 0,C 180,E1 -10709.998,E2 -10709.998} C_VEL
LIN {X 0,Y 411.212,Z 484.275,A -85,B 0,C 180,E1 -10710.817,E2 -10710.817} C_VEL
LIN {X 0,Y 410.595,Z 484.065,A -85,B 0,C 180,E1 -10711.637,E2 -10711.637} C_VEL
LIN {X 0,Y 407.801,Z 483.353,A -85,B 0,C 180,E1 -10712.969,E2 -10712.969} C_VEL
LIN {X 0,Y 405.085,Z 481.864,A -85,B 0,C 180,E1 -10714.302,E2 -10714.302} C_VEL
LIN {X 0,Y 404.6,Z 480.435,A -85,B 0,C 180,E1 -10715.112,E2 -10715.112} C_VEL
LIN {X 0,Y 404.795,Z 477.258,A -85,B 0,C 180,E1 -10716.477,E2 -10716.477} C_VEL
LIN {X 0,Y 405.452,Z 472.674,A -85,B 0,C 180,E1 -10717.968,E2 -10717.968} C_VEL
LIN {X 0,Y 405.953,Z 465.959,A -85,B 0,C 180,E1 -10719.69,E2 -10719.69} C_VEL
LIN {X 0,Y 406.521,Z 458.367,A -85,B 0,C 180,E1 -10721.212,E2 -10721.212} C_VEL
LIN {X 0,Y 407.211,Z 450.697,A -85,B 0,C 180,E1 -10722.456,E2 -10722.456} C_VEL
LIN {X 0,Y 407.88,Z 441.347,A -85,B 0,C 180,E1 -10723.702,E2 -10723.702} C_VEL
LIN {X 0,Y 408.519,Z 430.935,A -85,B 0,C 180,E1 -10724.824,E2 -10724.824} C_VEL
LIN {X 0,Y 409.124,Z 419.744,A -85,B 0,C 180,E1 -10725.773,E2 -10725.773} C_VEL
LIN {X 0,Y 409.666,Z 407.585,A -85,B 0,C 180,E1 -10726.568,E2 -10726.568} C_VEL
LIN {X 0,Y 409.924,Z 395.371,A -85,B 0,C 180,E1 -10727.158,E2 -10727.158} C_VEL
LIN {X 0,Y 409.65,Z 392.517,A -85,B 0,C 180,E1 -10727.281,E2 -10727.281} C_VEL
LIN {X 0,Y 405.662,Z 379.637,A -85,B 0,C 180,E1 -10727.852,E2 -10727.852} C_VEL
LIN {X 0,Y 405.514,Z 372.601,A -85,B 0,C 180,E1 -10730.628,E2 -10730.628} C_VEL
LIN {X 0,Y 405.474,Z 366.04,A -85,B 0,C 180,E1 -10733.491,E2 -10733.491} C_VEL
LIN {X 0,Y 405.48,Z 357.702,A -85,B 0,C 180,E1 -10737.325,E2 -10737.325} C_VEL
LIN {X 0,Y 405.627,Z 350.476,A -85,B 0,C 180,E1 -10740.735,E2 -10740.735} C_VEL
LIN {X 0,Y 405.767,Z 342.904,A -85,B 0,C 180,E1 -10744.253,E2 -10744.253} C_VEL
LIN {X 0,Y 405.473,Z 337.664,A -85,B 0,C 180,E1 -10746.587,E2 -10746.587} C_VEL
LIN {X 0,Y 404.144,Z 330.458,A -85,B 0,C 180,E1 -10749.8,E2 -10749.8} C_VEL
LIN {X 0,Y 404.136,Z 330.458,A -85,B 0,C 180,E1 -10753.081,E2 -10753.081} C_VEL
LIN {X 0,Y 404.187,Z 330.449,A -85,B 0,C 180,E1 -10755.931,E2 -10755.931} C_VEL
LIN {X 0,Y 404.15,Z 330.458,A -85,B 0,C 180,E1 -10758.638,E2 -10758.638} C_VEL
LIN {X 0,Y 404.146,Z 330.455,A -85,B 0,C 180,E1 -10761.488,E2 -10761.488} C_VEL
LIN {X 0,Y 404.167,Z 330.451,A -85,B 0,C 180,E1 -10764.982,E2 -10764.982} C_VEL
LIN {X 0,Y 404.122,Z 330.459,A -85,B 0,C 180,E1 -10768.552,E2 -10768.552} C_VEL
LIN {X 0,Y 404.175,Z 330.452,A -85,B 0,C 180,E1 -10771.998,E2 -10771.998} C_VEL
LIN {X 0,Y 404.159,Z 330.453,A -85,B 0,C 180,E1 -10775.333,E2 -10775.333} C_VEL
LIN {X 0,Y 404.18,Z 330.45,A -85,B 0,C 180,E1 -10778.582,E2 -10778.582} C_VEL
LIN {X 0,Y 404.191,Z 330.446,A -85,B 0,C 180,E1 -10781.761,E2 -10781.761} C_VEL
LIN {X 0,Y 404.185,Z 330.446,A -85,B 0,C 180,E1 -10784.881,E2 -10784.881} C_VEL
LIN {X 0,Y 404.252,Z 330.442,A -85,B 0,C 180,E1 -10787.958,E2 -10787.958} C_VEL
LIN {X 0,Y 404.409,Z 330.424,A -85,B 0,C 180,E1 -10792.099,E2 -10792.099} C_VEL
LIN {X 0,Y 404.401,Z 330.421,A -85,B 0,C 180,E1 -10794.014,E2 -10794.014} C_VEL
LIN {X 0,Y 404.454,Z 330.416,A -85,B 0,C 180,E1 -10798.008,E2 -10798.008} C_VEL
LIN {X 0,Y 404.585,Z 330.396,A -85,B 0,C 180,E1 -10800,E2 -10800} C_VEL
LIN {X 0,Y 404.41,Z 330.422,A -85,B 0,C 180,E1 -10802.988,E2 -10802.988} C_VEL
LIN {X 0,Y 404.416,Z 330.423,A -85,B 0,C 180,E1 -10805.985,E2 -10805.985} C_VEL
LIN {X 0,Y 404.398,Z 330.425,A -85,B 0,C 180,E1 -10807.991,E2 -10807.991} C_VEL
LIN {X 0,Y 404.247,Z 330.443,A -85,B 0,C 180,E1 -10812.041,E2 -10812.041} C_VEL
LIN {X 0,Y 404.188,Z 330.45,A -85,B 0,C 180,E1 -10815.118,E2 -10815.118} C_VEL
LIN {X 0,Y 404.192,Z 330.45,A -85,B 0,C 180,E1 -10818.238,E2 -10818.238} C_VEL
LIN {X 0,Y 404.178,Z 330.453,A -85,B 0,C 180,E1 -10821.417,E2 -10821.417} C_VEL
LIN {X 0,Y 404.156,Z 330.455,A -85,B 0,C 180,E1 -10824.667,E2 -10824.667} C_VEL
LIN {X 0,Y 404.172,Z 330.45,A -85,B 0,C 180,E1 -10828.001,E2 -10828.001} C_VEL
LIN {X 0,Y 404.117,Z 330.46,A -85,B 0,C 180,E1 -10831.559,E2 -10831.559} C_VEL
LIN {X 0,Y 404.164,Z 330.455,A -85,B 0,C 180,E1 -10835.018,E2 -10835.018} C_VEL
LIN {X 0,Y 404.138,Z 330.456,A -85,B 0,C 180,E1 -10838.758,E2 -10838.758} C_VEL
LIN {X 0,Y 404.183,Z 330.618,A -85,B 0,C 180,E1 -10839.154,E2 -10839.154} C_VEL
LIN {X 0,Y 407.074,Z 340.35,A -85,B 0,C 180,E1 -10842.324,E2 -10842.324} C_VEL
LIN {X 0,Y 410.747,Z 352.389,A -85,B 0,C 180,E1 -10845.941,E2 -10845.941} C_VEL
LIN {X 0,Y 413.983,Z 363.765,A -85,B 0,C 180,E1 -10849.064,E2 -10849.064} C_VEL
LIN {X 0,Y 416.71,Z 374.127,A -85,B 0,C 180,E1 -10851.702,E2 -10851.702} C_VEL
LIN {X 0,Y 416.585,Z 376.874,A -85,B 0,C 180,E1 -10852.302,E2 -10852.302} C_VEL
LIN {X 0,Y 413.814,Z 394.838,A -85,B 0,C 180,E1 -10855.916,E2 -10855.916} C_VEL
LIN {X 0,Y 411.64,Z 411.646,A -85,B 0,C 180,E1 -10859.193,E2 -10859.193} C_VEL
LIN {X 0,Y 410.963,Z 417.53,A -85,B 0,C 180,E1 -10860.317,E2 -10860.317} C_VEL
LIN {X 0,Y 415.507,Z 442.34,A -85,B 0,C 180,E1 -10861.209,E2 -10861.209} C_VEL
LIN {X 0,Y 417.877,Z 454.792,A -85,B 0,C 180,E1 -10861.787,E2 -10861.787} C_VEL
LIN {X 0,Y 416.851,Z 469.972,A -85,B 0,C 180,E1 -10862.42,E2 -10862.42} C_VEL
LIN {X 0,Y 415.489,Z 485.364,A -85,B 0,C 180,E1 -10863.236,E2 -10863.236} C_VEL
LIN {X 0,Y 414.086,Z 499.99,A -85,B 0,C 180,E1 -10864.203,E2 -10864.203} C_VEL
LIN {X 0,Y 412.528,Z 513.994,A -85,B 0,C 180,E1 -10865.333,E2 -10865.333} C_VEL
LIN {X 0,Y 410.889,Z 528.207,A -85,B 0,C 180,E1 -10866.704,E2 -10866.704} C_VEL
LIN {X 0,Y 409.27,Z 541.416,A -85,B 0,C 180,E1 -10868.216,E2 -10868.216} C_VEL
LIN {X 0,Y 407.791,Z 553.476,A -85,B 0,C 180,E1 -10869.84,E2 -10869.84} C_VEL
LIN {X 0,Y 406.513,Z 564.637,A -85,B 0,C 180,E1 -10871.611,E2 -10871.611} C_VEL
LIN {X 0,Y 405.407,Z 575.4,A -85,B 0,C 180,E1 -10873.641,E2 -10873.641} C_VEL
LIN {X 0,Y 404.426,Z 584.39,A -85,B 0,C 180,E1 -10875.665,E2 -10875.665} C_VEL
LIN {X 0,Y 403.909,Z 591.071,A -85,B 0,C 180,E1 -10877.441,E2 -10877.441} C_VEL
LIN {X 0,Y 403.435,Z 597.387,A -85,B 0,C 180,E1 -10879.463,E2 -10879.463} C_VEL
LIN {X 0,Y 403.209,Z 602.473,A -85,B 0,C 180,E1 -10881.483,E2 -10881.483} C_VEL
LIN {X 0,Y 403.124,Z 606.582,A -85,B 0,C 180,E1 -10883.576,E2 -10883.576} C_VEL
LIN {X 0,Y 403.004,Z 609.812,A -85,B 0,C 180,E1 -10886.003,E2 -10886.003} C_VEL
LIN {X 0,Y 403.037,Z 611.298,A -85,B 0,C 180,E1 -10888.004,E2 -10888.004} C_VEL
LIN {X 0,Y 402.991,Z 611.791,A -85,B 0,C 180,E1 -10890.002,E2 -10890.002} C_VEL
LIN {X 0,Y 403.049,Z 611.194,A -85,B 0,C 180,E1 -10892.001,E2 -10892.001} C_VEL
LIN {X 0,Y 403.009,Z 609.6,A -85,B 0,C 180,E1 -10894.002,E2 -10894.002} C_VEL
LIN {X 0,Y 403.166,Z 606.138,A -85,B 0,C 180,E1 -10896.476,E2 -10896.476} C_VEL
LIN {X 0,Y 403.263,Z 601.962,A -85,B 0,C 180,E1 -10898.521,E2 -10898.521} C_VEL
LIN {X 0,Y 403.454,Z 596.705,A -85,B 0,C 180,E1 -10900.541,E2 -10900.541} C_VEL
LIN {X 0,Y 403.968,Z 590.167,A -85,B 0,C 180,E1 -10902.563,E2 -10902.563} C_VEL
LIN {X 0,Y 404.564,Z 582.187,A -85,B 0,C 180,E1 -10904.592,E2 -10904.592} C_VEL
LIN {X 0,Y 405.482,Z 572.648,A -85,B 0,C 180,E1 -10906.62,E2 -10906.62} C_VEL
LIN {X 0,Y 406.439,Z 562.829,A -85,B 0,C 180,E1 -10908.397,E2 -10908.397} C_VEL
LIN {X 0,Y 407.742,Z 551.289,A -85,B 0,C 180,E1 -10910.167,E2 -10910.167} C_VEL
LIN {X 0,Y 409.137,Z 539.206,A -85,B 0,C 180,E1 -10911.748,E2 -10911.748} C_VEL
LIN {X 0,Y 410.736,Z 525.153,A -85,B 0,C 180,E1 -10913.311,E2 -10913.311} C_VEL
LIN {X 0,Y 412.378,Z 510.474,A -85,B 0,C 180,E1 -10914.682,E2 -10914.682} C_VEL
LIN {X 0,Y 413.991,Z 495.053,A -85,B 0,C 180,E1 -10915.877,E2 -10915.877} C_VEL
LIN {X 0,Y 415.409,Z 479.972,A -85,B 0,C 180,E1 -10916.842,E2 -10916.842} C_VEL
LIN {X 0,Y 416.729,Z 463.7,A -85,B 0,C 180,E1 -10917.673,E2 -10917.673} C_VEL
LIN {X 0,Y 417.279,Z 454.011,A -85,B 0,C 180,E1 -10918.079,E2 -10918.079} C_VEL
LIN {X 0,Y 414.363,Z 437.301,A -85,B 0,C 180,E1 -10918.877,E2 -10918.877} C_VEL
LIN {X 0,Y 411.59,Z 420.199,A -85,B 0,C 180,E1 -10919.528,E2 -10919.528} C_VEL
LIN {X 0,Y 410.663,Z 415.259,A -85,B 0,C 180,E1 -10919.757,E2 -10919.757} C_VEL
LIN {X 0,Y 412.599,Z 400.417,A -85,B 0,C 180,E1 -10922.741,E2 -10922.741} C_VEL
LIN {X 0,Y 414.994,Z 387.313,A -85,B 0,C 180,E1 -10925.621,E2 -10925.621} C_VEL
LIN {X 0,Y 417.359,Z 377.664,A -85,B 0,C 180,E1 -10927.956,E2 -10927.956} C_VEL
LIN {X 0,Y 417.512,Z 375.685,A -85,B 0,C 180,E1 -10928.524,E2 -10928.524} C_VEL
LIN {X 0,Y 416.676,Z 371.927,A -85,B 0,C 180,E1 -10929.864,E2 -10929.864} C_VEL
LIN {X 0,Y 415.315,Z 367.232,A -85,B 0,C 180,E1 -10931.878,E2 -10931.878} C_VEL
LIN {X 0,Y 414.005,Z 363.281,A -85,B 0,C 180,E1 -10934.109,E2 -10934.109} C_VEL
LIN {X 0,Y 413.232,Z 361.11,A -85,B 0,C 180,E1 -10935.789,E2 -10935.789} C_VEL
LIN {X 0,Y 412.747,Z 359.905,A -85,B 0,C 180,E1 -10937.071,E2 -10937.071} C_VEL
LIN {X 0,Y 411.966,Z 358.69,A -85,B 0,C 180,E1 -10939.589,E2 -10939.589} C_VEL
LIN {X 0,Y 411.464,Z 358.756,A -85,B 0,C 180,E1 -10942.056,E2 -10942.056} C_VEL
LIN {X 0,Y 410.684,Z 359.974,A -85,B 0,C 180,E1 -10944.42,E2 -10944.42} C_VEL
LIN {X 0,Y 409.729,Z 361.946,A -85,B 0,C 180,E1 -10946.71,E2 -10946.71} C_VEL
LIN {X 0,Y 408.543,Z 365.683,A -85,B 0,C 180,E1 -10950.075,E2 -10950.075} C_VEL
LIN {X 0,Y 407.647,Z 370.363,A -85,B 0,C 180,E1 -10953.705,E2 -10953.705} C_VEL
LIN {X 0,Y 407.146,Z 374.453,A -85,B 0,C 180,E1 -10956.609,E2 -10956.609} C_VEL
LIN {X 0,Y 406.668,Z 379.143,A -85,B 0,C 180,E1 -10959.657,E2 -10959.657} C_VEL
LIN {X 0,Y 411.71,Z 391.615,A -85,B 0,C 180,E1 -10960.794,E2 -10960.794} C_VEL
LIN {X 0,Y 414.233,Z 399.428,A -85,B 0,C 180,E1 -10961.502,E2 -10961.502} C_VEL
LIN {X 0,Y 414.253,Z 402.359,A -85,B 0,C 180,E1 -10961.7,E2 -10961.7} C_VEL
LIN {X 0,Y 412.963,Z 416.578,A -85,B 0,C 180,E1 -10962.709,E2 -10962.709} C_VEL
LIN {X 0,Y 411.815,Z 428.719,A -85,B 0,C 180,E1 -10963.773,E2 -10963.773} C_VEL
LIN {X 0,Y 410.644,Z 440.079,A -85,B 0,C 180,E1 -10964.998,E2 -10964.998} C_VEL
LIN {X 0,Y 409.576,Z 450.411,A -85,B 0,C 180,E1 -10966.353,E2 -10966.353} C_VEL
LIN {X 0,Y 408.582,Z 459.699,A -85,B 0,C 180,E1 -10967.836,E2 -10967.836} C_VEL
LIN {X 0,Y 407.666,Z 467.266,A -85,B 0,C 180,E1 -10969.32,E2 -10969.32} C_VEL
LIN {X 0,Y 406.695,Z 474.384,A -85,B 0,C 180,E1 -10971.053,E2 -10971.053} C_VEL
LIN {X 0,Y 406.128,Z 479.122,A -85,B 0,C 180,E1 -10972.543,E2 -10972.543} C_VEL
LIN {X 0,Y 405.581,Z 482.776,A -85,B 0,C 180,E1 -10974.033,E2 -10974.033} C_VEL
LIN {X 0,Y 405.446,Z 484.628,A -85,B 0,C 180,E1 -10975.028,E2 -10975.028} C_VEL
LIN {X 0,Y 405.205,Z 486.061,A -85,B 0,C 180,E1 -10976.022,E2 -10976.022} C_VEL
LIN {X 0,Y 404.999,Z 487.066,A -85,B 0,C 180,E1 -10977.016,E2 -10977.016} C_VEL
LIN {X 0,Y 404.76,Z 487.683,A -85,B 0,C 180,E1 -10978.01,E2 -10978.01} C_VEL
LIN {X 0,Y 404.637,Z 487.885,A -85,B 0,C 180,E1 -10979.005,E2 -10979.005} C_VEL
LIN {X 0,Y 404.522,Z 487.686,A -85,B 0,C 180,E1 -10980,E2 -10980} C_VEL
LIN {X 0,Y 404.486,Z 487.038,A -85,B 0,C 180,E1 -10980.996,E2 -10980.996} C_VEL
LIN {X 0,Y 404.396,Z 486,A -85,B 0,C 180,E1 -10981.992,E2 -10981.992} C_VEL
LIN {X 0,Y 404.517,Z 484.531,A -85,B 0,C 180,E1 -10982.988,E2 -10982.988} C_VEL
LIN {X 0,Y 404.482,Z 481.547,A -85,B 0,C 180,E1 -10984.485,E2 -10984.485} C_VEL
LIN {X 0,Y 404.564,Z 477.546,A -85,B 0,C 180,E1 -10985.983,E2 -10985.983} C_VEL
LIN {X 0,Y 405.03,Z 472.408,A -85,B 0,C 180,E1 -10987.478,E2 -10987.478} C_VEL
LIN {X 0,Y 405.426,Z 464.908,A -85,B 0,C 180,E1 -10989.227,E2 -10989.227} C_VEL
LIN {X 0,Y 405.899,Z 456.872,A -85,B 0,C 180,E1 -10990.728,E2 -10990.728} C_VEL
LIN {X 0,Y 406.416,Z 447.077,A -85,B 0,C 180,E1 -10992.23,E2 -10992.23} C_VEL
LIN {X 0,Y 407.154,Z 437.195,A -85,B 0,C 180,E1 -10993.476,E2 -10993.476} C_VEL
LIN {X 0,Y 407.848,Z 425.164,A -85,B 0,C 180,E1 -10994.725,E2 -10994.725} C_VEL
LIN {X 0,Y 408.463,Z 413.264,A -85,B 0,C 180,E1 -10995.732,E2 -10995.732} C_VEL
LIN {X 0,Y 409.226,Z 400.603,A -85,B 0,C 180,E1 -10996.59,E2 -10996.59} C_VEL
LIN {X 0,Y 409.565,Z 391.556,A -85,B 0,C 180,E1 -10997.088,E2 -10997.088} C_VEL
LIN {X 0,Y 406.27,Z 377.277,A -85,B 0,C 180,E1 -10997.875,E2 -10997.875} C_VEL
LIN {X 0,Y 403.903,Z 368.18,A -85,B 0,C 180,E1 -10998.286,E2 -10998.286} C_VEL
LIN {X 0,Y 404.076,Z 362.27,A -85,B 0,C 180,E1 -11001.423,E2 -11001.423} C_VEL
LIN {X 0,Y 404.247,Z 356.271,A -85,B 0,C 180,E1 -11004.661,E2 -11004.661} C_VEL
LIN {X 0,Y 404.561,Z 349.217,A -85,B 0,C 180,E1 -11008.538,E2 -11008.538} C_VEL
LIN {X 0,Y 404.775,Z 343.567,A -85,B 0,C 180,E1 -11011.702,E2 -11011.702} C_VEL
LIN {X 0,Y 404.943,Z 337.892,A -85,B 0,C 180,E1 -11014.941,E2 -11014.941} C_VEL
LIN {X 0,Y 404.666,Z 333.659,A -85,B 0,C 180,E1 -11017.435,E2 -11017.435} C_VEL
LIN {X 0,Y 404.181,Z 330.457,A -85,B 0,C 180,E1 -11019.396,E2 -11019.396} C_VEL
LIN {X 0,Y 404.159,Z 330.454,A -85,B 0,C 180,E1 -11023.082,E2 -11023.082} C_VEL
LIN {X 0,Y 404.157,Z 330.456,A -85,B 0,C 180,E1 -11025.925,E2 -11025.925} C_VEL
LIN {X 0,Y 404.122,Z 330.46,A -85,B 0,C 180,E1 -11028.633,E2 -11028.633} C_VEL
LIN {X 0,Y 404.195,Z 330.651,A -85,B 0,C 180,E1 -11030.443,E2 -11030.443} C_VEL
LIN {X 0,Y 405.417,Z 337.347,A -85,B 0,C 180,E1 -11033.416,E2 -11033.416} C_VEL
LIN {X 0,Y 405.765,Z 341.245,A -85,B 0,C 180,E1 -11035.138,E2 -11035.138} C_VEL
LIN {X 0,Y 405.601,Z 348.94,A -85,B 0,C 180,E1 -11038.678,E2 -11038.678} C_VEL
LIN {X 0,Y 405.479,Z 356.329,A -85,B 0,C 180,E1 -11042.125,E2 -11042.125} C_VEL
LIN {X 0,Y 405.414,Z 363.347,A -85,B 0,C 180,E1 -11045.413,E2 -11045.413} C_VEL
LIN {X 0,Y 405.481,Z 370.67,A -85,B 0,C 180,E1 -11048.653,E2 -11048.653} C_VEL
LIN {X 0,Y 405.688,Z 379.563,A -85,B 0,C 180,E1 -11052.225,E2 -11052.225} C_VEL
LIN {X 0,Y 409.94,Z 393.518,A -85,B 0,C 180,E1 -11052.869,E2 -11052.869} C_VEL
LIN {X 0,Y 409.652,Z 405.787,A -85,B 0,C 180,E1 -11053.426,E2 -11053.426} C_VEL
LIN {X 0,Y 409.252,Z 417.239,A -85,B 0,C 180,E1 -11054.138,E2 -11054.138} C_VEL
LIN {X 0,Y 408.673,Z 428.493,A -85,B 0,C 180,E1 -11055.049,E2 -11055.049} C_VEL
LIN {X 0,Y 408.03,Z 439.445,A -85,B 0,C 180,E1 -11056.171,E2 -11056.171} C_VEL
LIN {X 0,Y 407.46,Z 448.284,A -85,B 0,C 180,E1 -11057.294,E2 -11057.294} C_VEL
LIN {X 0,Y 406.549,Z 457.802,A -85,B 0,C 180,E1 -11058.784,E2 -11058.784} C_VEL
LIN {X 0,Y 405.966,Z 465.413,A -85,B 0,C 180,E1 -11060.281,E2 -11060.281} C_VEL
LIN {X 0,Y 405.583,Z 470.54,A -85,B 0,C 180,E1 -11061.528,E2 -11061.528} C_VEL
LIN {X 0,Y 405.081,Z 475.567,A -85,B 0,C 180,E1 -11063.022,E2 -11063.022} C_VEL
LIN {X 0,Y 404.72,Z 479.452,A -85,B 0,C 180,E1 -11064.517,E2 -11064.517} C_VEL
LIN {X 0,Y 404.535,Z 482.303,A -85,B 0,C 180,E1 -11066.013,E2 -11066.013} C_VEL
LIN {X 0,Y 404.443,Z 483.687,A -85,B 0,C 180,E1 -11067.009,E2 -11067.009} C_VEL
LIN {X 0,Y 404.212,Z 485.275,A -85,B 0,C 180,E1 -11069.001,E2 -11069.001} C_VEL
LIN {X 0,Y 404.196,Z 485.352,A -85,B 0,C 180,E1 -11070.831,E2 -11070.831} C_VEL
LIN {X 0,Y 404.301,Z 484.744,A -85,B 0,C 180,E1 -11071.99,E2 -11071.99} C_VEL
LIN {X 0,Y 404.456,Z 483.791,A -85,B 0,C 180,E1 -11072.986,E2 -11072.986} C_VEL
LIN {X 0,Y 404.555,Z 482.465,A -85,B 0,C 180,E1 -11073.982,E2 -11073.982} C_VEL
LIN {X 0,Y 404.6,Z 480.435,A -85,B 0,C 180,E1 -11075.112,E2 -11075.112} C_VEL
LIN {X 0,Y 404.154,Z 478.79,A -85,B 0,C 180,E1 -11075.914,E2 -11075.914} C_VEL
LIN {X 0,Y 401.655,Z 475.866,A -85,B 0,C 180,E1 -11077.218,E2 -11077.218} C_VEL
LIN {X 0,Y 399.209,Z 472.289,A -85,B 0,C 180,E1 -11078.497,E2 -11078.497} C_VEL
LIN {X 0,Y 398.848,Z 469.563,A -85,B 0,C 180,E1 -11079.249,E2 -11079.249} C_VEL
LIN {X 0,Y 399.43,Z 462.102,A -85,B 0,C 180,E1 -11080.9,E2 -11080.9} C_VEL
LIN {X 0,Y 400.232,Z 453.443,A -85,B 0,C 180,E1 -11082.419,E2 -11082.419} C_VEL
LIN {X 0,Y 400.973,Z 443.435,A -85,B 0,C 180,E1 -11083.813,E2 -11083.813} C_VEL
LIN {X 0,Y 401.644,Z 433.255,A -85,B 0,C 180,E1 -11084.954,E2 -11084.954} C_VEL
LIN {X 0,Y 402.364,Z 422.212,A -85,B 0,C 180,E1 -11085.934,E2 -11085.934} C_VEL
LIN {X 0,Y 402.843,Z 410.754,A -85,B 0,C 180,E1 -11086.727,E2 -11086.727} C_VEL
LIN {X 0,Y 403.216,Z 397.555,A -85,B 0,C 180,E1 -11087.404,E2 -11087.404} C_VEL
LIN {X 0,Y 402.983,Z 394.197,A -85,B 0,C 180,E1 -11087.549,E2 -11087.549} C_VEL
LIN {X 0,Y 399.277,Z 382.277,A -85,B 0,C 180,E1 -11088.102,E2 -11088.102} C_VEL
LIN {X 0,Y 398.796,Z 380.602,A -85,B 0,C 180,E1 -11088.183,E2 -11088.183} C_VEL
LIN {X 0,Y 398.58,Z 373.015,A -85,B 0,C 180,E1 -11091.201,E2 -11091.201} C_VEL
LIN {X 0,Y 398.536,Z 365.513,A -85,B 0,C 180,E1 -11094.479,E2 -11094.479} C_VEL
LIN {X 0,Y 398.581,Z 357.599,A -85,B 0,C 180,E1 -11098.16,E2 -11098.16} C_VEL
LIN {X 0,Y 398.709,Z 350.825,A -85,B 0,C 180,E1 -11101.328,E2 -11101.328} C_VEL
LIN {X 0,Y 398.83,Z 344.332,A -85,B 0,C 180,E1 -11104.321,E2 -11104.321} C_VEL
LIN {X 0,Y 398.683,Z 340.042,A -85,B 0,C 180,E1 -11106.265,E2 -11106.265} C_VEL
LIN {X 0,Y 397.639,Z 334.031,A -85,B 0,C 180,E1 -11108.952,E2 -11108.952} C_VEL
LIN {X 0,Y 397.077,Z 331.339,A -85,B 0,C 180,E1 -11110.213,E2 -11110.213} C_VEL
LIN {X 0,Y 397.088,Z 331.338,A -85,B 0,C 180,E1 -11113.646,E2 -11113.646} C_VEL
LIN {X 0,Y 397.145,Z 331.328,A -85,B 0,C 180,E1 -11116.51,E2 -11116.51} C_VEL
LIN {X 0,Y 397.109,Z 331.33,A -85,B 0,C 180,E1 -11119.548,E2 -11119.548} C_VEL
LIN {X 0,Y 397.082,Z 331.336,A -85,B 0,C 180,E1 -11122.788,E2 -11122.788} C_VEL
LIN {X 0,Y 397.1,Z 331.332,A -85,B 0,C 180,E1 -11126.28,E2 -11126.28} C_VEL
LIN {X 0,Y 397.085,Z 331.329,A -85,B 0,C 180,E1 -11130.133,E2 -11130.133} C_VEL
LIN {X 0,Y 397.174,Z 331.322,A -85,B 0,C 180,E1 -11132.608,E2 -11132.608} C_VEL
LIN {X 0,Y 397.121,Z 331.331,A -85,B 0,C 180,E1 -11135.981,E2 -11135.981} C_VEL
LIN {X 0,Y 397.136,Z 331.329,A -85,B 0,C 180,E1 -11139.271,E2 -11139.271} C_VEL
LIN {X 0,Y 397.159,Z 331.324,A -85,B 0,C 180,E1 -11142.843,E2 -11142.843} C_VEL
LIN {X 0,Y 397.203,Z 331.315,A -85,B 0,C 180,E1 -11146.678,E2 -11146.678} C_VEL
LIN {X 0,Y 397.21,Z 331.315,A -85,B 0,C 180,E1 -11149.808,E2 -11149.808} C_VEL
LIN {X 0,Y 397.34,Z 331.302,A -85,B 0,C 180,E1 -11152.887,E2 -11152.887} C_VEL
LIN {X 0,Y 397.231,Z 331.311,A -85,B 0,C 180,E1 -11154.924,E2 -11154.924} C_VEL
LIN {X 0,Y 397.423,Z 331.292,A -85,B 0,C 180,E1 -11157.973,E2 -11157.973} C_VEL
LIN {X 0,Y 397.554,Z 331.271,A -85,B 0,C 180,E1 -11160,E2 -11160} C_VEL
LIN {X 0,Y 397.368,Z 331.299,A -85,B 0,C 180,E1 -11163.041,E2 -11163.041} C_VEL
LIN {X 0,Y 397.365,Z 331.3,A -85,B 0,C 180,E1 -11166.091,E2 -11166.091} C_VEL
LIN {X 0,Y 397.353,Z 331.301,A -85,B 0,C 180,E1 -11168.134,E2 -11168.134} C_VEL
LIN {X 0,Y 397.206,Z 331.321,A -85,B 0,C 180,E1 -11172.258,E2 -11172.258} C_VEL
LIN {X 0,Y 397.16,Z 331.325,A -85,B 0,C 180,E1 -11175.392,E2 -11175.392} C_VEL
LIN {X 0,Y 397.15,Z 331.327,A -85,B 0,C 180,E1 -11178.574,E2 -11178.574} C_VEL
LIN {X 0,Y 397.153,Z 331.327,A -85,B 0,C 180,E1 -11181.815,E2 -11181.815} C_VEL
LIN {X 0,Y 397.13,Z 331.329,A -85,B 0,C 180,E1 -11185.514,E2 -11185.514} C_VEL
LIN {X 0,Y 397.099,Z 331.335,A -85,B 0,C 180,E1 -11188.545,E2 -11188.545} C_VEL
LIN {X 0,Y 397.056,Z 331.34,A -85,B 0,C 180,E1 -11192.073,E2 -11192.073} C_VEL
LIN {X 0,Y 397.099,Z 331.334,A -85,B 0,C 180,E1 -11195.505,E2 -11195.505} C_VEL
LIN {X 0,Y 397.105,Z 331.457,A -85,B 0,C 180,E1 -11198.337,E2 -11198.337} C_VEL
LIN {X 0,Y 400.671,Z 343.363,A -85,B 0,C 180,E1 -11202.296,E2 -11202.296} C_VEL
LIN {X 0,Y 404.3,Z 355.398,A -85,B 0,C 180,E1 -11205.951,E2 -11205.951} C_VEL
LIN {X 0,Y 407.434,Z 366.533,A -85,B 0,C 180,E1 -11209.048,E2 -11209.048} C_VEL
LIN {X 0,Y 410.033,Z 376.364,A -85,B 0,C 180,E1 -11211.591,E2 -11211.591} C_VEL
LIN {X 0,Y 409.495,Z 380.631,A -85,B 0,C 180,E1 -11212.502,E2 -11212.502} C_VEL
LIN {X 0,Y 406.816,Z 397.797,A -85,B 0,C 180,E1 -11216.019,E2 -11216.019} C_VEL
LIN {X 0,Y 404.512,Z 415.137,A -85,B 0,C 180,E1 -11219.46,E2 -11219.46} C_VEL
LIN {X 0,Y 404.257,Z 417.298,A -85,B 0,C 180,E1 -11219.869,E2 -11219.869} C_VEL
LIN {X 0,Y 408.769,Z 441.813,A -85,B 0,C 180,E1 -11220.768,E2 -11220.768} C_VEL
LIN {X 0,Y 411.335,Z 456.493,A -85,B 0,C 180,E1 -11221.459,E2 -11221.459} C_VEL
LIN {X 0,Y 410.116,Z 472.214,A -85,B 0,C 180,E1 -11222.153,E2 -11222.153} C_VEL
LIN {X 0,Y 408.635,Z 487.681,A -85,B 0,C 180,E1 -11223.027,E2 -11223.027} C_VEL
LIN {X 0,Y 407.112,Z 502.645,A -85,B 0,C 180,E1 -11224.082,E2 -11224.082} C_VEL
LIN {X 0,Y 405.411,Z 516.786,A -85,B 0,C 180,E1 -11225.281,E2 -11225.281} C_VEL
LIN {X 0,Y 403.765,Z 530.503,A -85,B 0,C 180,E1 -11226.675,E2 -11226.675} C_VEL
LIN {X 0,Y 402.064,Z 543.583,A -85,B 0,C 180,E1 -11228.259,E2 -11228.259} C_VEL
LIN {X 0,Y 400.539,Z 555.694,A -85,B 0,C 180,E1 -11229.995,E2 -11229.995} C_VEL
LIN {X 0,Y 399.149,Z 567.226,A -85,B 0,C 180,E1 -11231.952,E2 -11231.952} C_VEL
LIN {X 0,Y 398.175,Z 576.752,A -85,B 0,C 180,E1 -11233.862,E2 -11233.862} C_VEL
LIN {X 0,Y 397.338,Z 584.408,A -85,B 0,C 180,E1 -11235.666,E2 -11235.666} C_VEL
LIN {X 0,Y 396.734,Z 591.747,A -85,B 0,C 180,E1 -11237.729,E2 -11237.729} C_VEL
LIN {X 0,Y 396.284,Z 597.79,A -85,B 0,C 180,E1 -11239.787,E2 -11239.787} C_VEL
LIN {X 0,Y 396.127,Z 602.602,A -85,B 0,C 180,E1 -11241.843,E2 -11241.843} C_VEL
LIN {X 0,Y 396.071,Z 606.264,A -85,B 0,C 180,E1 -11243.891,E2 -11243.891} C_VEL
LIN {X 0,Y 395.969,Z 608.846,A -85,B 0,C 180,E1 -11245.931,E2 -11245.931} C_VEL
LIN {X 0,Y 396,Z 610.326,A -85,B 0,C 180,E1 -11247.968,E2 -11247.968} C_VEL
LIN {X 0,Y 395.959,Z 610.813,A -85,B 0,C 180,E1 -11250.002,E2 -11250.002} C_VEL
LIN {X 0,Y 396.015,Z 610.196,A -85,B 0,C 180,E1 -11252.036,E2 -11252.036} C_VEL
LIN {X 0,Y 395.978,Z 608.586,A -85,B 0,C 180,E1 -11254.073,E2 -11254.073} C_VEL
LIN {X 0,Y 396.129,Z 605.203,A -85,B 0,C 180,E1 -11256.522,E2 -11256.522} C_VEL
LIN {X 0,Y 396.206,Z 600.869,A -85,B 0,C 180,E1 -11258.674,E2 -11258.674} C_VEL
LIN {X 0,Y 396.435,Z 595.575,A -85,B 0,C 180,E1 -11260.73,E2 -11260.73} C_VEL
LIN {X 0,Y 396.942,Z 589.13,A -85,B 0,C 180,E1 -11262.748,E2 -11262.748} C_VEL
LIN {X 0,Y 397.464,Z 582.041,A -85,B 0,C 180,E1 -11264.596,E2 -11264.596} C_VEL
LIN {X 0,Y 398.402,Z 572.677,A -85,B 0,C 180,E1 -11266.66,E2 -11266.66} C_VEL
LIN {X 0,Y 399.565,Z 561.484,A -85,B 0,C 180,E1 -11268.726,E2 -11268.726} C_VEL
LIN {X 0,Y 400.89,Z 549.918,A -85,B 0,C 180,E1 -11270.527,E2 -11270.527} C_VEL
LIN {X 0,Y 402.509,Z 536.674,A -85,B 0,C 180,E1 -11272.271,E2 -11272.271} C_VEL
LIN {X 0,Y 404.021,Z 523.693,A -85,B 0,C 180,E1 -11273.722,E2 -11273.722} C_VEL
LIN {X 0,Y 405.781,Z 508.987,A -85,B 0,C 180,E1 -11275.11,E2 -11275.11} C_VEL
LIN {X 0,Y 407.475,Z 493.583,A -85,B 0,C 180,E1 -11276.319,E2 -11276.319} C_VEL
LIN {X 0,Y 408.885,Z 479.554,A -85,B 0,C 180,E1 -11277.237,E2 -11277.237} C_VEL
LIN {X 0,Y 410.347,Z 462.366,A -85,B 0,C 180,E1 -11278.133,E2 -11278.133} C_VEL
LIN {X 0,Y 410.718,Z 454.809,A -85,B 0,C 180,E1 -11278.467,E2 -11278.467} C_VEL
LIN {X 0,Y 408.179,Z 439.622,A -85,B 0,C 180,E1 -11279.24,E2 -11279.24} C_VEL
LIN {X 0,Y 405.647,Z 422.82,A -85,B 0,C 180,E1 -11279.931,E2 -11279.931} C_VEL
LIN {X 0,Y 404.054,Z 414.795,A -85,B 0,C 180,E1 -11280.295,E2 -11280.295} C_VEL
LIN {X 0,Y 406.374,Z 399.053,A -85,B 0,C 180,E1 -11283.604,E2 -11283.604} C_VEL
LIN {X 0,Y 408.51,Z 388.378,A -85,B 0,C 180,E1 -11286.043,E2 -11286.043} C_VEL
LIN {X 0,Y 410.685,Z 380.217,A -85,B 0,C 180,E1 -11288.077,E2 -11288.077} C_VEL
LIN {X 0,Y 410.943,Z 378.339,A -85,B 0,C 180,E1 -11288.627,E2 -11288.627} C_VEL
LIN {X 0,Y 409.956,Z 373.891,A -85,B 0,C 180,E1 -11290.271,E2 -11290.271} C_VEL
LIN {X 0,Y 408.668,Z 369.431,A -85,B 0,C 180,E1 -11292.313,E2 -11292.313} C_VEL
LIN {X 0,Y 407.868,Z 367.099,A -85,B 0,C 180,E1 -11293.639,E2 -11293.639} C_VEL
LIN {X 0,Y 406.63,Z 363.717,A -85,B 0,C 180,E1 -11296.264,E2 -11296.264} C_VEL
LIN {X 0,Y 405.982,Z 362.295,A -85,B 0,C 180,E1 -11298.108,E2 -11298.108} C_VEL
LIN {X 0,Y 405.417,Z 361.591,A -85,B 0,C 180,E1 -11300.104,E2 -11300.104} C_VEL
LIN {X 0,Y 404.755,Z 361.8,A -85,B 0,C 180,E1 -11302.575,E2 -11302.575} C_VEL
LIN {X 0,Y 403.895,Z 363.084,A -85,B 0,C 180,E1 -11304.955,E2 -11304.955} C_VEL
LIN {X 0,Y 402.856,Z 365.085,A -85,B 0,C 180,E1 -11307.262,E2 -11307.262} C_VEL
LIN {X 0,Y 401.565,Z 369.258,A -85,B 0,C 180,E1 -11311.057,E2 -11311.057} C_VEL
LIN {X 0,Y 400.829,Z 372.996,A -85,B 0,C 180,E1 -11314.002,E2 -11314.002} C_VEL
LIN {X 0,Y 400.187,Z 377.532,A -85,B 0,C 180,E1 -11317.272,E2 -11317.272} C_VEL
LIN {X 0,Y 399.98,Z 380.227,A -85,B 0,C 180,E1 -11319.02,E2 -11319.02} C_VEL
LIN {X 0,Y 405.787,Z 394.586,A -85,B 0,C 180,E1 -11320.424,E2 -11320.424} C_VEL
LIN {X 0,Y 408.185,Z 402.45,A -85,B 0,C 180,E1 -11321.176,E2 -11321.176} C_VEL
LIN {X 0,Y 406.812,Z 416.59,A -85,B 0,C 180,E1 -11322.179,E2 -11322.179} C_VEL
LIN {X 0,Y 405.444,Z 430.048,A -85,B 0,C 180,E1 -11323.381,E2 -11323.381} C_VEL
